  MoveL 1970 to (54.79, -51.67, -202.81) mm, rotated rx -11.83 ry -17.7 rz 126.62 deg; joints [4.443, -31.963, 116.112, 232.159, 70.658, -42.553, 143.741]
  MoveL 1971 to (53.18, -53.45, -205.23) mm, rotated rx -11.83 ry -17.7 rz 126.62 deg; joints [4.464, -31.726, 115.928, 232.166, 70.692, -42.511, 143.741]
  MoveL 1972 to (51.41, -54.45, -207.66) mm, rotated rx -11.83 ry -17.7 rz 126.62 deg; joints [4.497, -31.513, 115.805, 232.174, 70.75, -42.437, 143.741]
  MoveL 1973 to (50.67, -54.51, -208.61) mm, rotated rx -11.83 ry -17.7 rz 126.62 deg; joints [4.514, -31.44, 115.785, 232.177, 70.783, -42.394, 143.741]
  MoveL 1974 to (50.01, -54.27, -209.39) mm, rotated rx -11.83 ry -17.7 rz 126.62 deg; joints [4.532, -31.389, 115.791, 232.18, 70.82, -42.347, 143.741]
  MoveL 1975 to (49.72, -54.04, -209.71) mm, rotated rx -11.83 ry -17.7 rz 126.62 deg; joints [4.542, -31.372, 115.804, 232.181, 70.839, -42.322, 143.741]
  MoveL 1976 to (49.46, -53.74, -209.99) mm, rotated rx -11.83 ry -17.7 rz 126.62 deg; joints [4.551, -31.36, 115.824, 232.182, 70.859, -42.296, 143.741]
  MoveL 1977 to (48.99, -52.91, -210.43) mm, rotated rx -11.83 ry -17.7 rz 126.62 deg; joints [4.57, -31.353, 115.885, 232.183, 70.902, -42.242, 143.741]
  MoveL 1978 to (48.62, -51.78, -210.69) mm, rotated rx -11.83 ry -17.7 rz 126.62 deg; joints [4.59, -31.369, 115.972, 232.183, 70.948, -42.183, 143.741]
  MoveL 1979 to (48.34, -50.36, -210.77) mm, rotated rx -11.83 ry -17.7 rz 126.62 deg; joints [4.61, -31.406, 116.086, 232.182, 70.996, -42.12, 143.741]
  MoveL 1980 to (48.26, -49.84, -210.77) mm, rotated rx -11.83 ry -17.7 rz 126.62 deg; joints [4.616, -31.422, 116.128, 232.182, 71.013, -42.098, 143.741]
  MoveL 1981 to (48.22, -49.39, -210.74) mm, rotated rx -11.83 ry -17.7 rz 126.62 deg; joints [4.622, -31.438, 116.166, 232.182, 71.026, -42.081, 143.741]
  MoveL 1982 to (48.19, -48.96, -210.7) mm, rotated rx -11.83 ry -17.7 rz 126.62 deg; joints [4.627, -31.455, 116.201, 232.182, 71.038, -42.065, 143.741]
  MoveL 1983 to (48.17, -48.54, -210.64) mm, rotated rx -11.83 ry -17.7 rz 126.62 deg; joints [4.631, -31.472, 116.237, 232.181, 71.05, -42.05, 143.741]
  MoveL 1984 to (48.14, -48.09, -210.6) mm, rotated rx -11.83 ry -17.7 rz 126.62 deg; joints [4.636, -31.489, 116.274, 232.181, 71.062, -42.034, 143.741]
  MoveL 1985 to (48.07, -47.58, -210.58) mm, rotated rx -11.83 ry -17.7 rz 126.62 deg; joints [4.643, -31.506, 116.315, 232.181, 71.078, -42.013, 143.741]
  MoveL 1986 to (48, -47.06, -210.58) mm, rotated rx -11.83 ry -17.7 rz 126.62 deg; joints [4.649, -31.522, 116.357, 232.181, 71.095, -41.992, 143.741]
  MoveL 1987 to (47.93, -46.57, -210.58) mm, rotated rx -11.83 ry -17.7 rz 126.62 deg; joints [4.656, -31.538, 116.398, 232.18, 71.11, -41.972, 143.741]
  MoveL 1988 to (47.87, -46.1, -210.55) mm, rotated rx -11.83 ry -17.7 rz 126.62 deg; joints [4.662, -31.553, 116.436, 232.18, 71.124, -41.953, 143.741]
  MoveL 1989 to (47.84, -45.68, -210.5) mm, rotated rx -11.83 ry -17.7 rz 126.62 deg; joints [4.667, -31.57, 116.471, 232.181, 71.136, -41.938, 143.741]
  MoveL 1990 to (47.81, -45.25, -210.44) mm, rotated rx -11.83 ry -17.7 rz 126.62 deg; joints [4.672, -31.587, 116.506, 232.181, 71.147, -41.924, 143.741]
  MoveL 1991 to (47.77, -44.79, -210.38) mm, rotated rx -11.83 ry -17.7 rz 126.62 deg; joints [4.677, -31.606, 116.545, 232.181, 71.16, -41.907, 143.741]
  MoveL 1992 to (47.71, -44.18, -210.35) mm, rotated rx -11.83 ry -17.7 rz 126.62 deg; joints [4.685, -31.627, 116.595, 232.181, 71.178, -41.883, 143.741]
  MoveL 1993 to (47.63, -43.39, -210.33) mm, rotated rx -11.83 ry -17.7 rz 126.62 deg; joints [4.694, -31.653, 116.659, 232.18, 71.202, -41.852, 143.741]
  MoveL 1994 to (47.4, -41.84, -210.33) mm, rotated rx -11.83 ry -17.7 rz 126.62 deg; joints [4.715, -31.7, 116.785, 232.18, 71.252, -41.788, 143.741]
  MoveL 1995 to (47.29, -41.01, -210.3) mm, rotated rx -11.83 ry -17.7 rz 126.62 deg; joints [4.725, -31.728, 116.852, 232.18, 71.277, -41.755, 143.741]
  MoveL 1996 to (47.21, -40.39, -210.28) mm, rotated rx -11.83 ry -17.7 rz 126.62 deg; joints [4.733, -31.748, 116.903, 232.179, 71.296, -41.73, 143.741]
  MoveL 1997 to (47.19, -39.9, -210.28) mm, rotated rx -11.83 ry -17.7 rz 126.62 deg; joints [4.738, -31.764, 116.943, 232.178, 71.311, -41.71, 143.741]
  MoveL 1998 to (47.21, -39.48, -210.26) mm, rotated rx -11.83 ry -17.7 rz 126.62 deg; joints [4.74, -31.78, 116.978, 232.175, 71.323, -41.695, 143.741]
  MoveL 1999 to (47.26, -39.28, -210.15) mm, rotated rx -11.83 ry -17.7 rz 126.62 deg; joints [4.741, -31.794, 116.996, 232.175, 71.325, -41.691, 143.741]
  MoveL 2000 to (47.3, -39.34, -209.93) mm, rotated rx -11.83 ry -17.7 rz 126.62 deg; joints [4.742, -31.806, 116.993, 232.18, 71.316, -41.704, 143.741]
  MoveL 2001 to (47.32, -39.68, -209.58) mm, rotated rx -11.83 ry -17.7 rz 126.62 deg; joints [4.744, -31.814, 116.967, 232.191, 71.295, -41.733, 143.741]
  MoveL 2002 to (48.02, -39.34, -208.88) mm, rotated rx -11.83 ry -17.7 rz 126.62 deg; joints [4.726, -31.883, 117.01, 232.18, 71.278, -41.753, 143.741]
  MoveL 2003 to (48.92, -37.54, -208.73) mm, rotated rx -11.83 ry -17.7 rz 126.62 deg; joints [4.703, -31.975, 117.174, 232.138, 71.321, -41.692, 143.741]
  MoveL 2004 to (49.81, -35.84, -208.44) mm, rotated rx -11.83 ry -17.7 rz 126.62 deg; joints [4.682, -32.071, 117.33, 232.1, 71.357, -41.64, 143.741]
  MoveL 2005 to (50.69, -34.12, -208.17) mm, rotated rx -11.83 ry -17.7 rz 126.62 deg; joints [4.661, -32.166, 117.488, 232.062, 71.394, -41.587, 143.741]
  MoveL 2006 to (51.56, -32.39, -207.9) mm, rotated rx -11.83 ry -17.7 rz 126.62 deg; joints [4.641, -32.262, 117.646, 232.025, 71.431, -41.534, 143.741]
  MoveL 2007 to (52.46, -30.58, -207.68) mm, rotated rx -11.83 ry -17.7 rz 126.62 deg; joints [4.618, -32.358, 117.811, 231.984, 71.472, -41.476, 143.741]
  MoveL 2008 to (53.47, -28.71, -207.54) mm, rotated rx -11.83 ry -17.7 rz 126.62 deg; joints [4.591, -32.454, 117.981, 231.937, 71.516, -41.413, 143.741]
  MoveL 2009 to (54.76, -26.53, -207.43) mm, rotated rx -11.83 ry -17.7 rz 126.62 deg; joints [4.553, -32.566, 118.182, 231.875, 71.568, -41.337, 143.741]
  MoveL 2010 to (55.72, -24.23, -207.36) mm, rotated rx -11.83 ry -17.7 rz 126.62 deg; joints [4.53, -32.671, 118.386, 231.826, 71.628, -41.254, 143.741]
  MoveL 2011 to (56.53, -22.28, -207.24) mm, rotated rx -11.83 ry -17.7 rz 126.62 deg; joints [4.511, -32.764, 118.56, 231.785, 71.678, -41.186, 143.741]
  MoveL 2012 to (57.3, -20.55, -207.07) mm, rotated rx -11.83 ry -17.7 rz 126.62 deg; joints [4.493, -32.851, 118.715, 231.749, 71.718, -41.129, 143.741]
  MoveL 2013 to (58.17, -18.7, -206.94) mm, rotated rx -11.83 ry -17.7 rz 126.62 deg; joints [4.471, -32.942, 118.881, 231.708, 71.763, -41.066, 143.741]
  MoveL 2014 to (59.06, -16.82, -206.81) mm, rotated rx -11.83 ry -17.7 rz 126.62 deg; joints [4.448, -33.035, 119.05, 231.665, 71.809, -41.003, 143.741]
  MoveL 2015 to (59.99, -14.86, -206.74) mm, rotated rx -11.83 ry -17.7 rz 126.62 deg; joints [4.423, -33.128, 119.225, 231.618, 71.859, -40.933, 143.741]
  MoveL 2016 to (60.9, -12.92, -206.51) mm, rotated rx -11.83 ry -17.7 rz 126.62 deg; joints [4.401, -33.228, 119.398, 231.577, 71.903, -40.872, 143.741]
  MoveL 2017 to (61.8, -10.99, -206.4) mm, rotated rx -11.83 ry -17.7 rz 126.62 deg; joints [4.377, -33.322, 119.57, 231.533, 71.951, -40.806, 143.741]
  MoveL 2018 to (62.7, -9.06, -206.18) mm, rotated rx -11.83 ry -17.7 rz 126.62 deg; joints [4.356, -33.422, 119.743, 231.493, 71.995, -40.745, 143.741]
  MoveL 2019 to (63.6, -7.12, -206.07) mm, rotated rx -11.83 ry -17.7 rz 126.62 deg; joints [4.332, -33.515, 119.916, 231.449, 72.043, -40.68, 143.741]
  MoveL 2020 to (64.49, -5.18, -205.85) mm, rotated rx -11.83 ry -17.7 rz 126.62 deg; joints [4.311, -33.615, 120.088, 231.409, 72.088, -40.618, 143.741]
  MoveL 2021 to (65.39, -3.24, -205.74) mm, rotated rx -11.83 ry -17.7 rz 126.62 deg; joints [4.287, -33.708, 120.26, 231.365, 72.135, -40.553, 143.741]
  MoveL 2022 to (66.29, -1.3, -205.63) mm, rotated rx -11.83 ry -17.7 rz 126.62 deg; joints [4.263, -33.801, 120.432, 231.321, 72.184, -40.488, 143.741]
  MoveL 2023 to (67.04, 0.46, -205.4) mm, rotated rx -11.83 ry -17.7 rz 126.62 deg; joints [4.247, -33.891, 120.587, 231.288, 72.223, -40.434, 143.741]
  MoveL 2024 to (67.71, 2.16, -205.1) mm, rotated rx -11.83 ry -17.7 rz 126.62 deg; joints [4.233, -33.982, 120.737, 231.26, 72.259, -40.385, 143.741]
  MoveL 2025 to (68.34, 3.85, -204.71) mm, rotated rx -11.83 ry -17.7 rz 126.62 deg; joints [4.224, -34.077, 120.885, 231.237, 72.293, -40.341, 143.741]
  MoveL 2026 to (67.49, 2.71, -203.79) mm, rotated rx -11.83 ry -17.7 rz 126.62 deg; joints [4.266, -34.072, 120.784, 231.304, 72.234, -40.422, 143.741]
  MoveL 2027 to (67.66, 3.03, -203.73) mm, rotated rx -11.83 ry -17.7 rz 126.62 deg; joints [4.262, -34.091, 120.813, 231.297, 72.241, -40.413, 143.741]
  MoveL 2028 to (67.85, 3.35, -203.68) mm, rotated rx -11.83 ry -17.7 rz 126.62 deg; joints [4.256, -34.109, 120.842, 231.289, 72.247, -40.404, 143.741]
  MoveL 2029 to (68.13, 3.66, -203.64) mm, rotated rx -11.83 ry -17.7 rz 126.62 deg; joints [4.247, -34.129, 120.871, 231.277, 72.253, -40.396, 143.741]
  MoveL 2030 to (68.47, 3.95, -203.61) mm, rotated rx -11.83 ry -17.7 rz 126.62 deg; joints [4.234, -34.148, 120.9, 231.262, 72.258, -40.387, 143.741]
  MoveL 2031 to (68.89, 4.23, -203.61) mm, rotated rx -11.83 ry -17.7 rz 126.62 deg; joints [4.218, -34.168, 120.929, 231.244, 72.263, -40.38, 143.741]
  MoveL 2032 to (69.32, 4.5, -203.6) mm, rotated rx -11.83 ry -17.7 rz 126.62 deg; joints [4.202, -34.189, 120.958, 231.225, 72.267, -40.372, 143.741]
  MoveL 2033 to (70.23, 5.05, -203.6) mm, rotated rx -11.83 ry -17.7 rz 126.62 deg; joints [4.166, -34.229, 121.015, 231.185, 72.276, -40.357, 143.741]
  MoveL 2034 to (70.64, 5.31, -203.58) mm, rotated rx -11.83 ry -17.7 rz 126.62 deg; joints [4.15, -34.249, 121.042, 231.167, 72.28, -40.351, 143.741]
  MoveL 2035 to (71.03, 5.57, -203.54) mm, rotated rx -11.83 ry -17.7 rz 126.62 deg; joints [4.136, -34.27, 121.069, 231.151, 72.283, -40.346, 143.741]
  MoveL 2036 to (71.45, 5.88, -203.46) mm, rotated rx -11.83 ry -17.7 rz 126.62 deg; joints [4.121, -34.296, 121.101, 231.135, 72.286, -40.34, 143.741]
  MoveL 2037 to (71.92, 6.21, -203.39) mm, rotated rx -11.83 ry -17.7 rz 126.62 deg; joints [4.104, -34.323, 121.135, 231.115, 72.29, -40.333, 143.741]
  MoveL 2038 to (72.41, 6.53, -203.36) mm, rotated rx -11.83 ry -17.7 rz 126.62 deg; joints [4.086, -34.347, 121.167, 231.095, 72.294, -40.326, 143.741]
  MoveL 2039 to (72.87, 6.81, -203.35) mm, rotated rx -11.83 ry -17.7 rz 126.62 deg; joints [4.068, -34.368, 121.196, 231.075, 72.298, -40.319, 143.741]
  MoveL 2040 to (73.33, 7.08, -203.35) mm, rotated rx -11.83 ry -17.7 rz 126.62 deg; joints [4.05, -34.389, 121.225, 231.055, 72.303, -40.312, 143.741]
  MoveL 2041 to (74.23, 7.62, -203.35) mm, rotated rx -11.83 ry -17.7 rz 126.62 deg; joints [4.014, -34.429, 121.282, 231.015, 72.311, -40.297, 143.741]
  MoveL 2042 to (75.09, 8.17, -203.32) mm, rotated rx -11.83 ry -17.7 rz 126.62 deg; joints [3.981, -34.471, 121.339, 230.977, 72.32, -40.283, 143.741]
  MoveL 2043 to (77.35, 9.51, -203.32) mm, rotated rx -11.83 ry -17.7 rz 126.62 deg; joints [3.892, -34.571, 121.479, 230.878, 72.341, -40.248, 143.741]
  MoveL 2044 to (78.62, 10.19, -203.41) mm, rotated rx -11.83 ry -17.7 rz 126.62 deg; joints [3.84, -34.621, 121.551, 230.82, 72.353, -40.227, 143.741]
  MoveL 2045 to (79.73, 10.61, -203.67) mm, rotated rx -11.83 ry -17.7 rz 126.62 deg; joints [3.791, -34.646, 121.6, 230.765, 72.366, -40.207, 143.741]
  MoveL 2046 to (80.65, 10.77, -204.11) mm, rotated rx -11.83 ry -17.7 rz 126.62 deg; joints [3.746, -34.649, 121.623, 230.713, 72.377, -40.188, 143.741]
  MoveL 2047 to (81.05, 10.75, -204.39) mm, rotated rx -11.83 ry -17.7 rz 126.62 deg; joints [3.724, -34.641, 121.626, 230.689, 72.383, -40.179, 143.741]
  MoveL 2048 to (81.41, 10.67, -204.72) mm, rotated rx -11.83 ry -17.7 rz 126.62 deg; joints [3.703, -34.628, 121.623, 230.666, 72.389, -40.17, 143.741]
  MoveL 2049 to (81.98, 10.31, -205.51) mm, rotated rx -11.83 ry -17.7 rz 126.62 deg; joints [3.664, -34.583, 121.598, 230.621, 72.399, -40.153, 143.741]
  MoveL 2050 to (82.38, 9.68, -206.48) mm, rotated rx -11.83 ry -17.7 rz 126.62 deg; joints [3.629, -34.515, 121.549, 230.581, 72.41, -40.136, 143.741]
  MoveL 2051 to (82.66, 7.66, -208.93) mm, rotated rx -11.83 ry -17.7 rz 126.62 deg; joints [3.568, -34.309, 121.377, 230.511, 72.429, -40.107, 143.741]
  MoveL 2052 to (82.24, 5.27, -211.39) mm, rotated rx -11.83 ry -17.7 rz 126.62 deg; joints [3.535, -34.074, 121.165, 230.472, 72.443, -40.086, 143.741]
  MoveL 2053 to (81.1, 3.2, -213.14) mm, rotated rx -11.83 ry -17.7 rz 126.62 deg; joints [3.545, -33.874, 120.972, 230.481, 72.448, -40.081, 143.741]
  MoveL 2054 to (80.27, 2.28, -213.76) mm, rotated rx -11.83 ry -17.7 rz 126.62 deg; joints [3.567, -33.787, 120.883, 230.503, 72.448, -40.083, 143.741]
  MoveL 2055 to (79.26, 1.45, -214.2) mm, rotated rx -11.83 ry -17.7 rz 126.62 deg; joints [3.599, -33.708, 120.799, 230.537, 72.445, -40.089, 143.741]
  MoveL 2056 to (76.71, 0.01, -214.55) mm, rotated rx -11.83 ry -17.7 rz 126.62 deg; joints [3.695, -33.577, 120.645, 230.639, 72.434, -40.111, 143.741]
  MoveL 2057 to (74.29, -1.04, -214.54) mm, rotated rx -11.83 ry -17.7 rz 126.62 deg; joints [3.792, -33.483, 120.526, 230.744, 72.422, -40.135, 143.741]
  MoveL 2058 to (73.81, -1.24, -214.53) mm, rotated rx -11.83 ry -17.7 rz 126.62 deg; joints [3.812, -33.465, 120.502, 230.765, 72.419, -40.14, 143.741]
  MoveL 2059 to (73.31, -1.44, -214.5) mm, rotated rx -11.83 ry -17.7 rz 126.62 deg; joints [3.833, -33.448, 120.479, 230.787, 72.417, -40.145, 143.741]
  MoveL 2060 to (72.85, -1.63, -214.49) mm, rotated rx -11.83 ry -17.7 rz 126.62 deg; joints [3.851, -33.431, 120.457, 230.807, 72.414, -40.15, 143.741]
  MoveL 2061 to (72.44, -1.82, -214.51) mm, rotated rx -11.83 ry -17.7 rz 126.62 deg; joints [3.867, -33.413, 120.436, 230.824, 72.412, -40.154, 143.741]
  MoveL 2062 to (72, -2.03, -214.54) mm, rotated rx -11.83 ry -17.7 rz 126.62 deg; joints [3.884, -33.394, 120.412, 230.843, 72.41, -40.158, 143.741]
  MoveL 2063 to (71.49, -2.3, -214.61) mm, rotated rx -11.83 ry -17.7 rz 126.62 deg; joints [3.904, -33.368, 120.382, 230.863, 72.408, -40.162, 143.741]
  MoveL 2064 to (70.98, -2.58, -214.69) mm, rotated rx -11.83 ry -17.7 rz 126.62 deg; joints [3.922, -33.342, 120.352, 230.883, 72.407, -40.166, 143.741]
  MoveL 2065 to (70.48, -2.84, -214.73) mm, rotated rx -11.83 ry -17.7 rz 126.62 deg; joints [3.942, -33.318, 120.323, 230.904, 72.405, -40.17, 143.741]
  MoveL 2066 to (70, -3.07, -214.76) mm, rotated rx -11.83 ry -17.7 rz 126.62 deg; joints [3.961, -33.298, 120.298, 230.924, 72.402, -40.175, 143.741]
  MoveL 2067 to (69.52, -3.28, -214.77) mm, rotated rx -11.83 ry -17.7 rz 126.62 deg; joints [3.98, -33.278, 120.274, 230.944, 72.4, -40.18, 143.741]
  MoveL 2068 to (69.04, -3.49, -214.77) mm, rotated rx -11.83 ry -17.7 rz 126.62 deg; joints [3.999, -33.26, 120.25, 230.965, 72.397, -40.184, 143.741]
  MoveL 2069 to (68.54, -3.74, -214.8) mm, rotated rx -11.83 ry -17.7 rz 126.62 deg; joints [4.019, -33.237, 120.222, 230.986, 72.395, -40.189, 143.741]
  MoveL 2070 to (68.05, -4, -214.85) mm, rotated rx -11.83 ry -17.7 rz 126.62 deg; joints [4.037, -33.213, 120.193, 231.006, 72.393, -40.194, 143.741]
  MoveL 2071 to (67.57, -4.28, -214.92) mm, rotated rx -11.83 ry -17.7 rz 126.62 deg; joints [4.055, -33.188, 120.163, 231.025, 72.39, -40.199, 143.741]
  MoveL 2072 to (67.16, -4.58, -214.98) mm, rotated rx -11.83 ry -17.7 rz 126.62 deg; joints [4.07, -33.165, 120.132, 231.042, 72.386, -40.205, 143.741]
  MoveL 2073 to (66.81, -4.88, -215.01) mm, rotated rx -11.83 ry -17.7 rz 126.62 deg; joints [4.082, -33.144, 120.102, 231.057, 72.381, -40.214, 143.741]
  MoveL 2074 to (66.56, -5.19, -215.02) mm, rotated rx -11.83 ry -17.7 rz 126.62 deg; joints [4.091, -33.127, 120.073, 231.069, 72.373, -40.224, 143.741]
  MoveL 2075 to (66.33, -5.51, -215.02) mm, rotated rx -11.83 ry -17.7 rz 126.62 deg; joints [4.098, -33.111, 120.043, 231.08, 72.365, -40.235, 143.741]
  MoveL 2076 to (67.2, -4.56, -215.9) mm, rotated rx -11.83 ry -17.7 rz 126.62 deg; joints [4.055, -33.112, 120.129, 231.015, 72.417, -40.164, 143.741]
  MoveL 2077 to (66.44, -5.97, -216.18) mm, rotated rx -11.83 ry -17.7 rz 126.62 deg; joints [4.074, -33.031, 120.002, 231.046, 72.388, -40.203, 143.741]
  MoveL 2078 to (65.53, -7.53, -216.37) mm, rotated rx -11.83 ry -17.7 rz 126.62 deg; joints [4.099, -32.946, 119.86, 231.085, 72.354, -40.25, 143.741]
  MoveL 2079 to (64.47, -9.28, -216.51) mm, rotated rx -11.83 ry -17.7 rz 126.62 deg; joints [4.131, -32.854, 119.7, 231.135, 72.312, -40.307, 143.741]
  MoveL 2080 to (63.27, -11.18, -216.59) mm, rotated rx -11.83 ry -17.7 rz 126.62 deg; joints [4.169, -32.757, 119.526, 231.191, 72.266, -40.371, 143.741]
  MoveL 2081 to (62.15, -13, -216.74) mm, rotated rx -11.83 ry -17.7 rz 126.62 deg; joints [4.202, -32.661, 119.36, 231.242, 72.223, -40.429, 143.741]
  MoveL 2082 to (61.03, -14.82, -216.95) mm, rotated rx -11.83 ry -17.7 rz 126.62 deg; joints [4.234, -32.561, 119.193, 231.292, 72.183, -40.486, 143.741]
  MoveL 2083 to (59.96, -16.55, -217.08) mm, rotated rx -11.83 ry -17.7 rz 126.62 deg; joints [4.266, -32.47, 119.034, 231.341, 72.142, -40.543, 143.741]
  MoveL 2084 to (59.01, -18.13, -217.34) mm, rotated rx -11.83 ry -17.7 rz 126.62 deg; joints [4.292, -32.379, 118.888, 231.382, 72.109, -40.589, 143.741]
  MoveL 2085 to (57.92, -19.89, -217.56) mm, rotated rx -11.83 ry -17.7 rz 126.62 deg; joints [4.324, -32.282, 118.727, 231.429, 72.07, -40.643, 143.741]
  MoveL 2086 to (56.81, -21.65, -217.7) mm, rotated rx -11.83 ry -17.7 rz 126.62 deg; joints [4.357, -32.188, 118.564, 231.48, 72.029, -40.701, 143.741]
  MoveL 2087 to (55.66, -23.45, -217.8) mm, rotated rx -11.83 ry -17.7 rz 126.62 deg; joints [4.391, -32.094, 118.397, 231.534, 71.985, -40.762, 143.741]
  MoveL 2088 to (54.53, -25.25, -218.03) mm, rotated rx -11.83 ry -17.7 rz 126.62 deg; joints [4.423, -31.994, 118.231, 231.583, 71.946, -40.818, 143.741]
  MoveL 2089 to (53.37, -27.05, -218.29) mm, rotated rx -11.83 ry -17.7 rz 126.62 deg; joints [4.457, -31.89, 118.063, 231.633, 71.907, -40.873, 143.741]
  MoveL 2090 to (52.22, -28.84, -218.38) mm, rotated rx -11.83 ry -17.7 rz 126.62 deg; joints [4.491, -31.798, 117.897, 231.687, 71.864, -40.935, 143.741]
  MoveL 2091 to (51.05, -30.67, -218.42) mm, rotated rx -11.83 ry -17.7 rz 126.62 deg; joints [4.528, -31.705, 117.727, 231.744, 71.818, -41, 143.741]
  MoveL 2092 to (49.9, -32.45, -218.53) mm, rotated rx -11.83 ry -17.7 rz 126.62 deg; joints [4.562, -31.612, 117.562, 231.797, 71.775, -41.061, 143.741]
  MoveL 2093 to (48.75, -34.22, -218.73) mm, rotated rx -11.83 ry -17.7 rz 126.62 deg; joints [4.595, -31.513, 117.395, 231.848, 71.735, -41.119, 143.741]
  MoveL 2094 to (47.6, -35.96, -219.06) mm, rotated rx -11.83 ry -17.7 rz 126.62 deg; joints [4.627, -31.408, 117.232, 231.895, 71.701, -41.169, 143.741]
  MoveL 2095 to (46.4, -37.75, -219.32) mm, rotated rx -11.83 ry -17.7 rz 126.62 deg; joints [4.661, -31.304, 117.063, 231.947, 71.663, -41.224, 143.741]
  MoveL 2096 to (45.21, -39.52, -219.52) mm, rotated rx -11.83 ry -17.7 rz 126.62 deg; joints [4.695, -31.204, 116.896, 231.999, 71.624, -41.281, 143.741]
  MoveL 2097 to (43.98, -41.32, -219.76) mm, rotated rx -11.83 ry -17.7 rz 126.62 deg; joints [4.731, -31.1, 116.725, 232.052, 71.585, -41.339, 143.741]
  MoveL 2098 to (42.8, -43.11, -219.9) mm, rotated rx -11.83 ry -17.7 rz 126.62 deg; joints [4.766, -31.003, 116.556, 232.107, 71.543, -41.4, 143.741]
  MoveL 2099 to (41.65, -44.89, -219.93) mm, rotated rx -11.83 ry -17.7 rz 126.62 deg; joints [4.8, -30.914, 116.389, 232.163, 71.497, -41.467, 143.741]
  MoveL 2100 to (41.06, -45.13, -220.59) mm, rotated rx -11.83 ry -17.7 rz 126.62 deg; joints [4.814, -30.854, 116.356, 232.169, 71.515, -41.445, 143.741]
  MoveL 2101 to (41.16, -44.81, -220.92) mm, rotated rx -11.83 ry -17.7 rz 126.62 deg; joints [4.808, -30.848, 116.382, 232.154, 71.534, -41.418, 143.741]
  MoveL 2102 to (41.17, -44.77, -221.13) mm, rotated rx -11.83 ry -17.7 rz 126.62 deg; joints [4.805, -30.838, 116.385, 232.148, 71.541, -41.407, 143.741]
  MoveL 2103 to (41.1, -44.97, -221.23) mm, rotated rx -11.83 ry -17.7 rz 126.62 deg; joints [4.805, -30.824, 116.366, 232.15, 71.539, -41.411, 143.741]
  MoveL 2104 to (41.02, -45.39, -221.25) mm, rotated rx -11.83 ry -17.7 rz 126.62 deg; joints [4.805, -30.807, 116.33, 232.155, 71.527, -41.427, 143.741]
  MoveC 2105 to (40.97, -46.4, -221.25) mm, rotated rx -11.83 ry -17.7 rz 126.62 deg; joints [4.8, -30.771, 116.245, 232.162, 71.496, -41.468, 143.741] to (41, -47.42, -221.25) mm, rotated rx -11.83 ry -17.7 rz 126.62 deg; joints [4.792, -30.738, 116.16, 232.168, 71.464, -41.51, 143.741]
  MoveL 2106 to (41, -47.42, -221.25) mm, rotated rx -11.83 ry -17.7 rz 126.62 deg; joints [4.792, -30.737, 116.16, 232.167, 71.464, -41.51, 143.741]
  MoveL 2107 to (41, -47.96, -221.28) mm, rotated rx -11.83 ry -17.7 rz 126.62 deg; joints [4.787, -30.718, 116.115, 232.17, 71.448, -41.531, 143.741]
  MoveL 2108 to (40.98, -48.5, -221.33) mm, rotated rx -11.83 ry -17.7 rz 126.62 deg; joints [4.784, -30.696, 116.069, 232.173, 71.433, -41.551, 143.741]
  MoveL 2109 to (40.95, -49.08, -221.4) mm, rotated rx -11.83 ry -17.7 rz 126.62 deg; joints [4.78, -30.672, 116.02, 232.176, 71.417, -41.572, 143.741]
  MoveL 2110 to (40.93, -49.68, -221.44) mm, rotated rx -11.83 ry -17.7 rz 126.62 deg; joints [4.776, -30.65, 115.97, 232.179, 71.4, -41.595, 143.741]
  MoveL 2111 to (40.94, -50.89, -221.46) mm, rotated rx -11.83 ry -17.7 rz 126.62 deg; joints [4.767, -30.608, 115.868, 232.185, 71.363, -41.644, 143.741]
  MoveL 2112 to (40.93, -51.45, -221.49) mm, rotated rx -11.83 ry -17.7 rz 126.62 deg; joints [4.763, -30.587, 115.821, 232.188, 71.347, -41.665, 143.741]
  MoveL 2113 to (40.89, -51.92, -221.56) mm, rotated rx -11.83 ry -17.7 rz 126.62 deg; joints [4.76, -30.566, 115.781, 232.191, 71.335, -41.682, 143.741]
  MoveL 2114 to (40.85, -52.35, -221.65) mm, rotated rx -11.83 ry -17.7 rz 126.62 deg; joints [4.757, -30.545, 115.743, 232.193, 71.324, -41.695, 143.741]
  MoveL 2115 to (40.82, -52.78, -221.72) mm, rotated rx -11.83 ry -17.7 rz 126.62 deg; joints [4.755, -30.526, 115.707, 232.195, 71.313, -41.71, 143.741]
  MoveL 2116 to (40.81, -53.23, -221.75) mm, rotated rx -11.83 ry -17.7 rz 126.62 deg; joints [4.752, -30.509, 115.669, 232.197, 71.3, -41.727, 143.741]
  MoveL 2117 to (40.86, -55.85, -221.75) mm, rotated rx -11.83 ry -17.7 rz 126.62 deg; joints [4.731, -30.421, 115.45, 232.211, 71.219, -41.835, 143.741]
  MoveL 2118 to (40.66, -58.75, -222.1) mm, rotated rx -11.83 ry -17.7 rz 126.62 deg; joints [4.714, -30.298, 115.201, 232.228, 71.14, -41.939, 143.741]
  MoveL 2119 to (40.35, -59.99, -222.53) mm, rotated rx -11.83 ry -17.7 rz 126.62 deg; joints [4.713, -30.224, 115.089, 232.237, 71.117, -41.971, 143.741]
  MoveL 2120 to (39.89, -61.1, -223.13) mm, rotated rx -11.83 ry -17.7 rz 126.62 deg; joints [4.715, -30.142, 114.985, 232.245, 71.104, -41.989, 143.741]
  MoveL 2121 to (39.3, -62.07, -223.91) mm, rotated rx -11.83 ry -17.7 rz 126.62 deg; joints [4.722, -30.051, 114.889, 232.254, 71.101, -41.994, 143.741]
  MoveL 2122 to (38.57, -62.9, -224.86) mm, rotated rx -11.83 ry -17.7 rz 126.62 deg; joints [4.734, -29.952, 114.802, 232.262, 71.109, -41.985, 143.741]
  MoveL 2123 to (36.7, -64.16, -227.27) mm, rotated rx -11.83 ry -17.7 rz 126.62 deg; joints [4.77, -29.729, 114.65, 232.279, 71.155, -41.927, 143.741]
  MoveL 2124 to (34.85, -64.63, -229.68) mm, rotated rx -11.83 ry -17.7 rz 126.62 deg; joints [4.809, -29.534, 114.566, 232.29, 71.226, -41.837, 143.741]
  MoveL 2125 to (34.16, -64.47, -230.63) mm, rotated rx -11.83 ry -17.7 rz 126.62 deg; joints [4.826, -29.47, 114.561, 232.291, 71.264, -41.788, 143.741]
  MoveL 2126 to (33.62, -64.06, -231.41) mm, rotated rx -11.83 ry -17.7 rz 126.62 deg; joints [4.841, -29.427, 114.582, 232.289, 71.303, -41.736, 143.741]
  MoveL 2127 to (33.41, -63.75, -231.73) mm, rotated rx -11.83 ry -17.7 rz 126.62 deg; joints [4.847, -29.414, 114.602, 232.286, 71.324, -41.709, 143.741]
  MoveL 2128 to (33.24, -63.38, -232.01) mm, rotated rx -11.83 ry -17.7 rz 126.62 deg; joints [4.853, -29.407, 114.629, 232.283, 71.345, -41.681, 143.741]
  MoveL 2129 to (33.01, -62.45, -232.44) mm, rotated rx -11.83 ry -17.7 rz 126.62 deg; joints [4.863, -29.408, 114.7, 232.275, 71.389, -41.623, 143.741]
  MoveL 2130 to (32.94, -61.26, -232.7) mm, rotated rx -11.83 ry -17.7 rz 126.62 deg; joints [4.871, -29.432, 114.798, 232.263, 71.434, -41.562, 143.741]
  MoveL 2131 to (33.02, -59.81, -232.79) mm, rotated rx -11.83 ry -17.7 rz 126.62 deg; joints [4.877, -29.478, 114.92, 232.249, 71.482, -41.498, 143.741]
  MoveL 2132 to (33.07, -59.29, -232.79) mm, rotated rx -11.83 ry -17.7 rz 126.62 deg; joints [4.879, -29.496, 114.965, 232.243, 71.498, -41.476, 143.741]
  MoveL 2133 to (33.13, -58.84, -232.75) mm, rotated rx -11.83 ry -17.7 rz 126.62 deg; joints [4.88, -29.515, 115.004, 232.239, 71.51, -41.459, 143.741]
  MoveL 2134 to (33.21, -58.43, -232.7) mm, rotated rx -11.83 ry -17.7 rz 126.62 deg; joints [4.88, -29.533, 115.04, 232.235, 71.521, -41.445, 143.741]
  MoveL 2135 to (33.29, -58.03, -232.63) mm, rotated rx -11.83 ry -17.7 rz 126.62 deg; joints [4.88, -29.553, 115.075, 232.231, 71.531, -41.431, 143.741]
  MoveL 2136 to (33.37, -57.59, -232.58) mm, rotated rx -11.83 ry -17.7 rz 126.62 deg; joints [4.881, -29.572, 115.114, 232.227, 71.543, -41.415, 143.741]
  MoveL 2137 to (33.43, -57.09, -232.56) mm, rotated rx -11.83 ry -17.7 rz 126.62 deg; joints [4.882, -29.591, 115.157, 232.222, 71.558, -41.395, 143.741]
  MoveL 2138 to (34, -51.39, -232.55) mm, rotated rx -11.83 ry -17.7 rz 126.62 deg; joints [4.9, -29.795, 115.644, 232.165, 71.732, -41.161, 143.741]
  MoveL 2139 to (34.09, -50.63, -232.54) mm, rotated rx -11.83 ry -17.7 rz 126.62 deg; joints [4.901, -29.823, 115.709, 232.157, 71.755, -41.13, 143.741]
  MoveL 2140 to (34.19, -49.98, -232.53) mm, rotated rx -11.83 ry -17.7 rz 126.62 deg; joints [4.902, -29.847, 115.765, 232.149, 71.774, -41.104, 143.741]
  MoveL 2141 to (34.37, -49.43, -232.52) mm, rotated rx -11.83 ry -17.7 rz 126.62 deg; joints [4.898, -29.87, 115.814, 232.139, 71.79, -41.082, 143.741]
  MoveL 2142 to (34.61, -48.95, -232.48) mm, rotated rx -11.83 ry -17.7 rz 126.62 deg; joints [4.893, -29.895, 115.858, 232.128, 71.802, -41.065, 143.741]
  MoveL 2143 to (34.8, -48.68, -232.32) mm, rotated rx -11.83 ry -17.7 rz 126.62 deg; joints [4.889, -29.917, 115.885, 232.123, 71.804, -41.061, 143.741]
  MoveL 2144 to (34.82, -48.69, -232.01) mm, rotated rx -11.83 ry -17.7 rz 126.62 deg; joints [4.892, -29.935, 115.886, 232.131, 71.795, -41.075, 143.741]
  MoveL 2145 to (34.65, -49.02, -231.53) mm, rotated rx -11.83 ry -17.7 rz 126.62 deg; joints [4.904, -29.948, 115.86, 232.152, 71.771, -41.108, 143.741]
  MoveL 2146 to (35.27, -49.11, -230.55) mm, rotated rx -11.83 ry -17.7 rz 126.62 deg; joints [4.89, -30.015, 115.869, 232.154, 71.735, -41.156, 143.741]
  MoveL 2147 to (36.49, -47.69, -230.25) mm, rotated rx -11.83 ry -17.7 rz 126.62 deg; joints [4.854, -30.109, 116.009, 232.105, 71.761, -41.116, 143.741]
  MoveL 2148 to (37.77, -46.2, -230.05) mm, rotated rx -11.83 ry -17.7 rz 126.62 deg; joints [4.814, -30.201, 116.156, 232.051, 71.792, -41.069, 143.741]
  MoveL 2149 to (39.13, -44.57, -229.92) mm, rotated rx -11.83 ry -17.7 rz 126.62 deg; joints [4.77, -30.295, 116.315, 231.99, 71.83, -41.013, 143.741]
  MoveL 2150 to (41.85, -41.28, -229.92) mm, rotated rx -11.83 ry -17.7 rz 126.62 deg; joints [4.68, -30.47, 116.633, 231.862, 71.913, -40.891, 143.741]
  MoveL 2151 to (43.11, -39.75, -229.83) mm, rotated rx -11.83 ry -17.7 rz 126.62 deg; joints [4.639, -30.556, 116.781, 231.804, 71.949, -40.838, 143.741]
  MoveL 2152 to (44.47, -38.1, -229.83) mm, rotated rx -11.83 ry -17.7 rz 126.62 deg; joints [4.594, -30.644, 116.939, 231.74, 71.991, -40.777, 143.741]
  MoveL 2153 to (45.92, -36.5, -229.83) mm, rotated rx -11.83 ry -17.7 rz 126.62 deg; joints [4.544, -30.732, 117.095, 231.673, 72.03, -40.719, 143.741]
  MoveL 2154 to (47.65, -34.64, -229.65) mm, rotated rx -11.83 ry -17.7 rz 126.62 deg; joints [4.486, -30.846, 117.278, 231.597, 72.07, -40.66, 143.741]
  MoveL 2155 to (48.97, -32.84, -229.42) mm, rotated rx -11.83 ry -17.7 rz 126.62 deg; joints [4.447, -30.95, 117.449, 231.54, 72.11, -40.603, 143.741]
  MoveL 2156 to (50.27, -31.11, -229.3) mm, rotated rx -11.83 ry -17.7 rz 126.62 deg; joints [4.405, -31.046, 117.614, 231.481, 72.151, -40.545, 143.741]
  MoveL 2157 to (51.63, -29.46, -229.19) mm, rotated rx -11.83 ry -17.7 rz 126.62 deg; joints [4.361, -31.139, 117.772, 231.419, 72.189, -40.49, 143.741]
  MoveL 2158 to (52.98, -27.81, -228.98) mm, rotated rx -11.83 ry -17.7 rz 126.62 deg; joints [4.318, -31.239, 117.931, 231.361, 72.224, -40.44, 143.741]
  MoveL 2159 to (54.33, -26.16, -228.87) mm, rotated rx -11.83 ry -17.7 rz 126.62 deg; joints [4.273, -31.332, 118.089, 231.3, 72.263, -40.385, 143.741]
  MoveL 2160 to (55.68, -24.51, -228.76) mm, rotated rx -11.83 ry -17.7 rz 126.62 deg; joints [4.229, -31.425, 118.246, 231.239, 72.301, -40.331, 143.741]
  MoveL 2161 to (57.02, -22.85, -228.55) mm, rotated rx -11.83 ry -17.7 rz 126.62 deg; joints [4.186, -31.524, 118.405, 231.181, 72.336, -40.28, 143.741]
  MoveL 2162 to (58.37, -21.19, -228.44) mm, rotated rx -11.83 ry -17.7 rz 126.62 deg; joints [4.141, -31.617, 118.562, 231.12, 72.375, -40.226, 143.741]
  MoveL 2163 to (59.71, -19.54, -228.34) mm, rotated rx -11.83 ry -17.7 rz 126.62 deg; joints [4.097, -31.71, 118.719, 231.059, 72.413, -40.172, 143.741]
  MoveL 2164 to (61.04, -17.87, -228.13) mm, rotated rx -11.83 ry -17.7 rz 126.62 deg; joints [4.054, -31.809, 118.878, 231.002, 72.449, -40.122, 143.741]
  MoveL 2165 to (62.39, -16.21, -228.03) mm, rotated rx -11.83 ry -17.7 rz 126.62 deg; joints [4.009, -31.902, 119.035, 230.941, 72.488, -40.068, 143.741]
  MoveL 2166 to (63.49, -14.72, -227.77) mm, rotated rx -11.83 ry -17.7 rz 126.62 deg; joints [3.976, -31.992, 119.174, 230.895, 72.518, -40.027, 143.741]
  MoveL 2167 to (64.44, -13.35, -227.41) mm, rotated rx -11.83 ry -17.7 rz 126.62 deg; joints [3.949, -32.081, 119.303, 230.858, 72.542, -39.994, 143.741]
  MoveL 2168 to (65.25, -12.06, -226.9) mm, rotated rx -11.83 ry -17.7 rz 126.62 deg; joints [3.931, -32.173, 119.425, 230.832, 72.56, -39.969, 143.741]
  MoveL 2169 to (64.35, -12.75, -226.06) mm, rotated rx -11.83 ry -17.7 rz 126.62 deg; joints [3.977, -32.178, 119.36, 230.896, 72.517, -40.027, 143.741]
  MoveL 2170 to (64.56, -12.5, -226.03) mm, rotated rx -11.83 ry -17.7 rz 126.62 deg; joints [3.97, -32.193, 119.383, 230.886, 72.523, -40.02, 143.741]
  MoveL 2171 to (64.79, -12.27, -225.99) mm, rotated rx -11.83 ry -17.7 rz 126.62 deg; joints [3.962, -32.208, 119.406, 230.877, 72.527, -40.014, 143.741]
  MoveL 2172 to (65.1, -12.08, -225.93) mm, rotated rx -11.83 ry -17.7 rz 126.62 deg; joints [3.95, -32.225, 119.427, 230.865, 72.529, -40.011, 143.741]
  MoveL 2173 to (65.48, -11.9, -225.9) mm, rotated rx -11.83 ry -17.7 rz 126.62 deg; joints [3.936, -32.243, 119.447, 230.849, 72.53, -40.008, 143.741]
  MoveL 2174 to (65.94, -11.73, -225.87) mm, rotated rx -11.83 ry -17.7 rz 126.62 deg; joints [3.918, -32.261, 119.467, 230.831, 72.531, -40.005, 143.741]
  MoveL 2175 to (70.45, -10.38, -225.87) mm, rotated rx -11.83 ry -17.7 rz 126.62 deg; joints [3.733, -32.416, 119.644, 230.639, 72.537, -39.982, 143.741]
  MoveL 2176 to (70.83, -10.25, -225.85) mm, rotated rx -11.83 ry -17.7 rz 126.62 deg; joints [3.718, -32.431, 119.661, 230.623, 72.538, -39.98, 143.741]
  MoveL 2177 to (71.33, -10.1, -225.85) mm, rotated rx -11.83 ry -17.7 rz 126.62 deg; joints [3.697, -32.448, 119.68, 230.602, 72.539, -39.978, 143.741]
  MoveL 2178 to (72.31, -9.78, -225.81) mm, rotated rx -11.83 ry -17.7 rz 126.62 deg; joints [3.658, -32.485, 119.721, 230.561, 72.539, -39.974, 143.741]
  MoveL 2179 to (74.82, -9.03, -225.81) mm, rotated rx -11.83 ry -17.7 rz 126.62 deg; joints [3.555, -32.571, 119.818, 230.455, 72.543, -39.961, 143.741]
  MoveL 2180 to (75.79, -8.67, -225.79) mm, rotated rx -11.83 ry -17.7 rz 126.62 deg; joints [3.516, -32.607, 119.86, 230.414, 72.545, -39.955, 143.741]
  MoveL 2181 to (77.17, -8.24, -225.86) mm, rotated rx -11.83 ry -17.7 rz 126.62 deg; joints [3.458, -32.651, 119.915, 230.353, 72.55, -39.945, 143.741]
  MoveL 2182 to (78.32, -8.03, -226.11) mm, rotated rx -11.83 ry -17.7 rz 126.62 deg; joints [3.406, -32.672, 119.946, 230.298, 72.555, -39.934, 143.741]
  MoveL 2183 to (79.25, -8.04, -226.55) mm, rotated rx -11.83 ry -17.7 rz 126.62 deg; joints [3.36, -32.668, 119.956, 230.248, 72.562, -39.922, 143.741]
  MoveL 2184 to (79.63, -8.13, -226.84) mm, rotated rx -11.83 ry -17.7 rz 126.62 deg; joints [3.339, -32.657, 119.952, 230.225, 72.565, -39.916, 143.741]
  MoveL 2185 to (79.95, -8.27, -227.17) mm, rotated rx -11.83 ry -17.7 rz 126.62 deg; joints [3.319, -32.641, 119.943, 230.203, 72.569, -39.909, 143.741]
  MoveL 2186 to (80.43, -8.72, -227.99) mm, rotated rx -11.83 ry -17.7 rz 126.62 deg; joints [3.284, -32.59, 119.908, 230.164, 72.578, -39.896, 143.741]
  MoveL 2187 to (80.68, -9.39, -228.98) mm, rotated rx -11.83 ry -17.7 rz 126.62 deg; joints [3.254, -32.516, 119.85, 230.13, 72.588, -39.881, 143.741]
  MoveL 2188 to (80.51, -11.4, -231.54) mm, rotated rx -11.83 ry -17.7 rz 126.62 deg; joints [3.212, -32.296, 119.667, 230.079, 72.61, -39.85, 143.741]
  MoveL 2189 to (79.58, -13.61, -234.11) mm, rotated rx -11.83 ry -17.7 rz 126.62 deg; joints [3.202, -32.05, 119.456, 230.06, 72.631, -39.822, 143.741]
  MoveL 2190 to (78.02, -15.35, -235.94) mm, rotated rx -11.83 ry -17.7 rz 126.62 deg; joints [3.232, -31.848, 119.279, 230.084, 72.649, -39.803, 143.741]
  MoveL 2191 to (77, -16.04, -236.58) mm, rotated rx -11.83 ry -17.7 rz 126.62 deg; joints [3.262, -31.764, 119.204, 230.112, 72.656, -39.796, 143.741]
  MoveL 2192 to (75.83, -16.61, -237.04) mm, rotated rx -11.83 ry -17.7 rz 126.62 deg; joints [3.302, -31.69, 119.138, 230.151, 72.662, -39.791, 143.741]
  MoveL 2193 to (73.02, -17.39, -237.4) mm, rotated rx -11.83 ry -17.7 rz 126.62 deg; joints [3.412, -31.574, 119.031, 230.26, 72.671, -39.788, 143.741]
  MoveL 2194 to (69.92, -17.93, -237.4) mm, rotated rx -11.83 ry -17.7 rz 126.62 deg; joints [3.542, -31.481, 118.942, 230.39, 72.678, -39.788, 143.741]
  MoveL 2195 to (68.92, -18.13, -237.42) mm, rotated rx -11.83 ry -17.7 rz 126.62 deg; joints [3.583, -31.45, 118.911, 230.431, 72.68, -39.789, 143.741]
  MoveL 2196 to (67.89, -18.31, -237.42) mm, rotated rx -11.83 ry -17.7 rz 126.62 deg; joints [3.626, -31.419, 118.881, 230.474, 72.682, -39.789, 143.741]
  MoveL 2197 to (67.4, -18.4, -237.42) mm, rotated rx -11.83 ry -17.7 rz 126.62 deg; joints [3.646, -31.403, 118.866, 230.494, 72.683, -39.789, 143.741]
  MoveL 2198 to (66.75, -18.52, -237.45) mm, rotated rx -11.83 ry -17.7 rz 126.62 deg; joints [3.673, -31.382, 118.846, 230.521, 72.685, -39.789, 143.741]
  MoveL 2199 to (66.17, -18.66, -237.51) mm, rotated rx -11.83 ry -17.7 rz 126.62 deg; joints [3.696, -31.36, 118.826, 230.544, 72.687, -39.788, 143.741]
  MoveL 2200 to (65.68, -18.79, -237.58) mm, rotated rx -11.83 ry -17.7 rz 126.62 deg; joints [3.715, -31.34, 118.808, 230.562, 72.689, -39.787, 143.741]
  MoveL 2201 to (65.23, -18.9, -237.63) mm, rotated rx -11.83 ry -17.7 rz 126.62 deg; joints [3.733, -31.322, 118.792, 230.58, 72.691, -39.786, 143.741]
  MoveL 2202 to (64.78, -19, -237.67) mm, rotated rx -11.83 ry -17.7 rz 126.62 deg; joints [3.751, -31.306, 118.777, 230.598, 72.692, -39.786, 143.741]
  MoveL 2203 to (63.23, -19.27, -237.67) mm, rotated rx -11.83 ry -17.7 rz 126.62 deg; joints [3.816, -31.259, 118.731, 230.663, 72.695, -39.787, 143.741]
  MoveL 2204 to (62.74, -19.38, -237.68) mm, rotated rx -11.83 ry -17.7 rz 126.62 deg; joints [3.836, -31.243, 118.715, 230.683, 72.696, -39.787, 143.741]
  MoveL 2205 to (62.31, -19.49, -237.71) mm, rotated rx -11.83 ry -17.7 rz 126.62 deg; joints [3.853, -31.227, 118.699, 230.7, 72.696, -39.788, 143.741]
  MoveL 2206 to (61.95, -19.62, -237.75) mm, rotated rx -11.83 ry -17.7 rz 126.62 deg; joints [3.867, -31.211, 118.683, 230.715, 72.696, -39.789, 143.741]
  MoveL 2207 to (61.69, -19.78, -237.82) mm, rotated rx -11.83 ry -17.7 rz 126.62 deg; joints [3.876, -31.196, 118.665, 230.724, 72.695, -39.791, 143.741]
  MoveL 2208 to (61.48, -19.96, -237.89) mm, rotated rx -11.83 ry -17.7 rz 126.62 deg; joints [3.882, -31.181, 118.647, 230.732, 72.693, -39.794, 143.741]
  MoveL 2209 to (62.99, -19.46, -238.69) mm, rotated rx -11.83 ry -17.7 rz 126.62 deg; joints [3.81, -31.187, 118.705, 230.646, 72.724, -39.749, 143.741]
  MoveL 2210 to (61.69, -20.65, -239.1) mm, rotated rx -11.83 ry -17.7 rz 126.62 deg; joints [3.852, -31.093, 118.584, 230.695, 72.708, -39.773, 143.741]
  MoveL 2211 to (60.33, -21.94, -239.36) mm, rotated rx -11.83 ry -17.7 rz 126.62 deg; joints [3.898, -31.003, 118.456, 230.75, 72.686, -39.805, 143.741]
  MoveL 2212 to (58.89, -23.33, -239.54) mm, rotated rx -11.83 ry -17.7 rz 126.62 deg; joints [3.947, -30.913, 118.318, 230.812, 72.657, -39.845, 143.741]
  MoveL 2213 to (57.37, -24.83, -239.74) mm, rotated rx -11.83 ry -17.7 rz 126.62 deg; joints [3.999, -30.817, 118.17, 230.877, 72.627, -39.888, 143.741]
  MoveL 2214 to (55.84, -26.32, -239.83) mm, rotated rx -11.83 ry -17.7 rz 126.62 deg; joints [4.053, -30.726, 118.024, 230.945, 72.593, -39.936, 143.741]
  MoveL 2215 to (54.31, -27.8, -239.93) mm, rotated rx -11.83 ry -17.7 rz 126.62 deg; joints [4.107, -30.635, 117.877, 231.013, 72.56, -39.983, 143.741]
  MoveL 2216 to (52.78, -29.3, -240.13) mm, rotated rx -11.83 ry -17.7 rz 126.62 deg; joints [4.159, -30.538, 117.729, 231.078, 72.529, -40.027, 143.741]
  MoveL 2217 to (51.24, -30.78, -240.23) mm, rotated rx -11.83 ry -17.7 rz 126.62 deg; joints [4.213, -30.448, 117.581, 231.146, 72.496, -40.074, 143.741]
  MoveL 2218 to (49.71, -32.26, -240.33) mm, rotated rx -11.83 ry -17.7 rz 126.62 deg; joints [4.266, -30.357, 117.434, 231.214, 72.463, -40.122, 143.741]
  MoveL 2219 to (48.17, -33.74, -240.53) mm, rotated rx -11.83 ry -17.7 rz 126.62 deg; joints [4.318, -30.26, 117.286, 231.279, 72.433, -40.166, 143.741]
  MoveL 2220 to (45.09, -36.7, -240.73) mm, rotated rx -11.83 ry -17.7 rz 126.62 deg; joints [4.425, -30.078, 116.991, 231.415, 72.366, -40.263, 143.741]
  MoveL 2221 to (43.8, -37.93, -240.94) mm, rotated rx -11.83 ry -17.7 rz 126.62 deg; joints [4.468, -29.994, 116.866, 231.469, 72.342, -40.298, 143.741]
  MoveL 2222 to (42.41, -39.32, -241.01) mm, rotated rx -11.83 ry -17.7 rz 126.62 deg; joints [4.516, -29.912, 116.728, 231.531, 72.31, -40.345, 143.741]
  MoveL 2223 to (40.99, -40.81, -241.02) mm, rotated rx -11.83 ry -17.7 rz 126.62 deg; joints [4.565, -29.828, 116.581, 231.596, 72.273, -40.399, 143.741]
  MoveL 2224 to (39.05, -42.65, -241.13) mm, rotated rx -11.83 ry -17.7 rz 126.62 deg; joints [4.632, -29.715, 116.396, 231.682, 72.231, -40.461, 143.741]
  MoveL 2225 to (37.1, -44.34, -241.22) mm, rotated rx -11.83 ry -17.7 rz 126.62 deg; joints [4.701, -29.608, 116.222, 231.767, 72.194, -40.518, 143.741]
  MoveL 2226 to (35.47, -45.83, -241.32) mm, rotated rx -11.83 ry -17.7 rz 126.62 deg; joints [4.757, -29.514, 116.07, 231.839, 72.16, -40.568, 143.741]
  MoveL 2227 to (33.98, -47.23, -241.49) mm, rotated rx -11.83 ry -17.7 rz 126.62 deg; joints [4.807, -29.422, 115.928, 231.903, 72.131, -40.612, 143.741]
  MoveL 2228 to (32.58, -48.52, -241.77) mm, rotated rx -11.83 ry -17.7 rz 126.62 deg; joints [4.853, -29.33, 115.794, 231.959, 72.108, -40.648, 143.741]
  MoveL 2229 to (31.18, -49.8, -242.06) mm, rotated rx -11.83 ry -17.7 rz 126.62 deg; joints [4.898, -29.238, 115.662, 232.015, 72.085, -40.683, 143.741]
  MoveL 2230 to (29.77, -51.05, -242.35) mm, rotated rx -11.83 ry -17.7 rz 126.62 deg; joints [4.944, -29.147, 115.532, 232.071, 72.064, -40.717, 143.741]
  MoveL 2231 to (28.31, -52.39, -242.51) mm, rotated rx -11.83 ry -17.7 rz 126.62 deg; joints [4.993, -29.058, 115.393, 232.133, 72.035, -40.761, 143.741]
  MoveL 2232 to (27.66, -52.39, -243.13) mm, rotated rx -11.83 ry -17.7 rz 126.62 deg; joints [5.011, -29.007, 115.378, 232.143, 72.058, -40.732, 143.741]
  MoveL 2233 to (27.77, -52.09, -243.44) mm, rotated rx -11.83 ry -17.7 rz 126.62 deg; joints [5.005, -29.002, 115.403, 232.129, 72.076, -40.707, 143.741]
  MoveL 2234 to (27.74, -52.05, -243.63) mm, rotated rx -11.83 ry -17.7 rz 126.62 deg; joints [5.004, -28.992, 115.404, 232.125, 72.083, -40.697, 143.741]
  MoveL 2235 to (27.6, -52.26, -243.73) mm, rotated rx -11.83 ry -17.7 rz 126.62 deg; joints [5.007, -28.976, 115.383, 232.129, 72.08, -40.701, 143.741]
  MoveL 2236 to (27.42, -52.67, -243.75) mm, rotated rx -11.83 ry -17.7 rz 126.62 deg; joints [5.011, -28.957, 115.346, 232.138, 72.069, -40.717, 143.741]
  MoveL 2237 to (27.26, -53.13, -243.75) mm, rotated rx -11.83 ry -17.7 rz 126.62 deg; joints [5.014, -28.938, 115.305, 232.147, 72.056, -40.736, 143.741]
  MoveL 2238 to (27.05, -54.08, -243.78) mm, rotated rx -11.83 ry -17.7 rz 126.62 deg; joints [5.016, -28.9, 115.221, 232.16, 72.028, -40.774, 143.741]
  MoveL 2239 to (26.71, -55.62, -243.78) mm, rotated rx -11.83 ry -17.7 rz 126.62 deg; joints [5.019, -28.842, 115.087, 232.183, 71.981, -40.837, 143.741]
  MoveL 2240 to (26.46, -56.56, -243.8) mm, rotated rx -11.83 ry -17.7 rz 126.62 deg; joints [5.022, -28.804, 115.003, 232.198, 71.953, -40.875, 143.741]
  MoveL 2241 to (26.24, -57.59, -243.8) mm, rotated rx -11.83 ry -17.7 rz 126.62 deg; joints [5.024, -28.765, 114.913, 232.213, 71.922, -40.917, 143.741]
  MoveL 2242 to (26.12, -58.09, -243.82) mm, rotated rx -11.83 ry -17.7 rz 126.62 deg; joints [5.025, -28.745, 114.869, 232.22, 71.908, -40.938, 143.741]
  MoveL 2243 to (26, -58.55, -243.85) mm, rotated rx -11.83 ry -17.7 rz 126.62 deg; joints [5.026, -28.726, 114.829, 232.226, 71.895, -40.955, 143.741]
  MoveL 2244 to (25.89, -58.97, -243.89) mm, rotated rx -11.83 ry -17.7 rz 126.62 deg; joints [5.027, -28.706, 114.791, 232.232, 71.883, -40.971, 143.741]
  MoveL 2245 to (25.77, -59.36, -243.95) mm, rotated rx -11.83 ry -17.7 rz 126.62 deg; joints [5.028, -28.687, 114.756, 232.238, 71.874, -40.984, 143.741]
  MoveL 2246 to (25.66, -59.76, -244.01) mm, rotated rx -11.83 ry -17.7 rz 126.62 deg; joints [5.029, -28.668, 114.72, 232.243, 71.863, -40.998, 143.741]
  MoveL 2247 to (25.54, -60.21, -244.04) mm, rotated rx -11.83 ry -17.7 rz 126.62 deg; joints [5.03, -28.649, 114.68, 232.25, 71.851, -41.015, 143.741]
  MoveL 2248 to (25.42, -60.67, -244.07) mm, rotated rx -11.83 ry -17.7 rz 126.62 deg; joints [5.031, -28.63, 114.639, 232.257, 71.838, -41.033, 143.741]
  MoveL 2249 to (25.3, -61.09, -244.11) mm, rotated rx -11.83 ry -17.7 rz 126.62 deg; joints [5.033, -28.61, 114.601, 232.263, 71.826, -41.049, 143.741]
  MoveL 2250 to (25.18, -61.47, -244.17) mm, rotated rx -11.83 ry -17.7 rz 126.62 deg; joints [5.034, -28.591, 114.566, 232.269, 71.817, -41.062, 143.741]
  MoveL 2251 to (25.06, -61.86, -244.22) mm, rotated rx -11.83 ry -17.7 rz 126.62 deg; joints [5.036, -28.573, 114.531, 232.274, 71.807, -41.076, 143.741]
  MoveL 2252 to (24.94, -62.29, -244.25) mm, rotated rx -11.83 ry -17.7 rz 126.62 deg; joints [5.037, -28.554, 114.493, 232.281, 71.795, -41.092, 143.741]
  MoveL 2253 to (24.83, -62.8, -244.25) mm, rotated rx -11.83 ry -17.7 rz 126.62 deg; joints [5.038, -28.535, 114.448, 232.288, 71.779, -41.114, 143.741]
  MoveL 2254 to (23.95, -65.58, -244.61) mm, rotated rx -11.83 ry -17.7 rz 126.62 deg; joints [5.049, -28.402, 114.196, 232.331, 71.707, -41.213, 143.741]
  MoveL 2255 to (23.38, -66.74, -245.05) mm, rotated rx -11.83 ry -17.7 rz 126.62 deg; joints [5.059, -28.325, 114.085, 232.349, 71.687, -41.242, 143.741]
  MoveL 2256 to (22.7, -67.73, -245.68) mm, rotated rx -11.83 ry -17.7 rz 126.62 deg; joints [5.071, -28.241, 113.985, 232.366, 71.678, -41.256, 143.741]
  MoveL 2257 to (21.07, -69.24, -247.46) mm, rotated rx -11.83 ry -17.7 rz 126.62 deg; joints [5.103, -28.052, 113.816, 232.393, 71.692, -41.241, 143.741]
  MoveL 2258 to (19.06, -70.11, -249.95) mm, rotated rx -11.83 ry -17.7 rz 126.62 deg; joints [5.146, -27.835, 113.687, 232.413, 71.748, -41.169, 143.741]
  MoveL 2259 to (17.27, -70.21, -252.44) mm, rotated rx -11.83 ry -17.7 rz 126.62 deg; joints [5.185, -27.648, 113.626, 232.42, 71.827, -41.066, 143.741]
  MoveL 2260 to (16.67, -69.93, -253.42) mm, rotated rx -11.83 ry -17.7 rz 126.62 deg; joints [5.198, -27.587, 113.631, 232.417, 71.868, -41.012, 143.741]
  MoveL 2261 to (16.28, -69.43, -254.22) mm, rotated rx -11.83 ry -17.7 rz 126.62 deg; joints [5.207, -27.549, 113.659, 232.408, 71.909, -40.957, 143.741]
  MoveL 2262 to (16.16, -69.1, -254.56) mm, rotated rx -11.83 ry -17.7 rz 126.62 deg; joints [5.21, -27.538, 113.683, 232.403, 71.93, -40.929, 143.741]
  MoveL 2263 to (16.09, -68.71, -254.85) mm, rotated rx -11.83 ry -17.7 rz 126.62 deg; joints [5.212, -27.533, 113.712, 232.396, 71.951, -40.9, 143.741]
  MoveL 2264 to (16.1, -67.76, -255.29) mm, rotated rx -11.83 ry -17.7 rz 126.62 deg; joints [5.213, -27.539, 113.788, 232.378, 71.994, -40.842, 143.741]
  MoveL 2265 to (16.31, -66.59, -255.56) mm, rotated rx -11.83 ry -17.7 rz 126.62 deg; joints [5.209, -27.567, 113.888, 232.356, 72.038, -40.781, 143.741]
  MoveL 2266 to (16.73, -65.2, -255.65) mm, rotated rx -11.83 ry -17.7 rz 126.62 deg; joints [5.201, -27.617, 114.012, 232.328, 72.082, -40.72, 143.741]
  MoveL 2267 to (17.58, -62.72, -255.65) mm, rotated rx -11.83 ry -17.7 rz 126.62 deg; joints [5.184, -27.717, 114.235, 232.28, 72.157, -40.617, 143.741]
  MoveL 2268 to (17.73, -62.31, -255.62) mm, rotated rx -11.83 ry -17.7 rz 126.62 deg; joints [5.181, -27.736, 114.273, 232.272, 72.168, -40.601, 143.741]
  MoveL 2269 to (17.89, -61.94, -255.57) mm, rotated rx -11.83 ry -17.7 rz 126.62 deg; joints [5.178, -27.755, 114.307, 232.265, 72.178, -40.588, 143.741]
  MoveL 2270 to (18.04, -61.59, -255.5) mm, rotated rx -11.83 ry -17.7 rz 126.62 deg; joints [5.175, -27.774, 114.34, 232.258, 72.186, -40.576, 143.741]
  MoveL 2271 to (18.21, -61.19, -255.45) mm, rotated rx -11.83 ry -17.7 rz 126.62 deg; joints [5.172, -27.793, 114.377, 232.251, 72.196, -40.562, 143.741]
  MoveL 2272 to (18.39, -60.72, -255.41) mm, rotated rx -11.83 ry -17.7 rz 126.62 deg; joints [5.168, -27.815, 114.419, 232.242, 72.209, -40.544, 143.741]
  MoveL 2273 to (18.59, -60.24, -255.35) mm, rotated rx -11.83 ry -17.7 rz 126.62 deg; joints [5.164, -27.838, 114.464, 232.233, 72.222, -40.526, 143.741]
  MoveL 2274 to (18.77, -59.73, -255.34) mm, rotated rx -11.83 ry -17.7 rz 126.62 deg; joints [5.16, -27.86, 114.51, 232.223, 72.237, -40.506, 143.741]
  MoveL 2275 to (18.98, -59.12, -255.35) mm, rotated rx -11.83 ry -17.7 rz 126.62 deg; joints [5.156, -27.884, 114.565, 232.211, 72.255, -40.48, 143.741]
  MoveL 2276 to (19.23, -58.29, -255.42) mm, rotated rx -11.83 ry -17.7 rz 126.62 deg; joints [5.151, -27.913, 114.638, 232.194, 72.282, -40.443, 143.741]
  MoveL 2277 to (19.4, -57.79, -255.42) mm, rotated rx -11.83 ry -17.7 rz 126.62 deg; joints [5.147, -27.933, 114.683, 232.184, 72.297, -40.423, 143.741]
  MoveL 2278 to (19.57, -57.32, -255.41) mm, rotated rx -11.83 ry -17.7 rz 126.62 deg; joints [5.144, -27.952, 114.725, 232.175, 72.311, -40.403, 143.741]
  MoveL 2279 to (19.73, -56.88, -255.39) mm, rotated rx -11.83 ry -17.7 rz 126.62 deg; joints [5.141, -27.972, 114.765, 232.167, 72.324, -40.386, 143.741]
  MoveL 2280 to (19.89, -56.5, -255.34) mm, rotated rx -11.83 ry -17.7 rz 126.62 deg; joints [5.138, -27.991, 114.801, 232.159, 72.334, -40.373, 143.741]
  MoveL 2281 to (20.06, -56.14, -255.28) mm, rotated rx -11.83 ry -17.7 rz 126.62 deg; joints [5.134, -28.01, 114.834, 232.152, 72.342, -40.36, 143.741]
  MoveL 2282 to (20.28, -55.78, -255.23) mm, rotated rx -11.83 ry -17.7 rz 126.62 deg; joints [5.128, -28.029, 114.869, 232.143, 72.351, -40.348, 143.741]
  MoveL 2283 to (20.53, -55.45, -255.17) mm, rotated rx -11.83 ry -17.7 rz 126.62 deg; joints [5.121, -28.049, 114.901, 232.132, 72.359, -40.337, 143.741]
  MoveL 2284 to (20.71, -55.32, -255.01) mm, rotated rx -11.83 ry -17.7 rz 126.62 deg; joints [5.117, -28.067, 114.917, 232.128, 72.357, -40.339, 143.741]
  MoveL 2285 to (20.71, -55.43, -254.7) mm, rotated rx -11.83 ry -17.7 rz 126.62 deg; joints [5.12, -28.081, 114.91, 232.137, 72.344, -40.356, 143.741]
  MoveL 2286 to (20.51, -55.82, -254.21) mm, rotated rx -11.83 ry -17.7 rz 126.62 deg; joints [5.133, -28.092, 114.878, 232.16, 72.319, -40.392, 143.741]
  MoveL 2287 to (21.19, -55.25, -253.35) mm, rotated rx -11.83 ry -17.7 rz 126.62 deg; joints [5.12, -28.175, 114.945, 232.152, 72.308, -40.406, 143.741]
  MoveL 2288 to (24.59, -52.67, -253.35) mm, rotated rx -11.83 ry -17.7 rz 126.62 deg; joints [4.997, -28.341, 115.22, 232, 72.37, -40.31, 143.741]
  MoveL 2289 to (26.18, -51.46, -253.29) mm, rotated rx -11.83 ry -17.7 rz 126.62 deg; joints [4.94, -28.422, 115.349, 231.931, 72.397, -40.269, 143.741]
  MoveL 2290 to (27.78, -50.27, -253.14) mm, rotated rx -11.83 ry -17.7 rz 126.62 deg; joints [4.884, -28.507, 115.477, 231.863, 72.421, -40.232, 143.741]
  MoveL 2291 to (29.62, -48.9, -252.94) mm, rotated rx -11.83 ry -17.7 rz 126.62 deg; joints [4.82, -28.607, 115.624, 231.787, 72.448, -40.19, 143.741]
  MoveL 2292 to (31.36, -47.6, -252.73) mm, rotated rx -11.83 ry -17.7 rz 126.62 deg; joints [4.759, -28.703, 115.764, 231.715, 72.472, -40.152, 143.741]
  MoveL 2293 to (33.1, -46.28, -252.63) mm, rotated rx -11.83 ry -17.7 rz 126.62 deg; joints [4.697, -28.793, 115.904, 231.64, 72.501, -40.109, 143.741]
  MoveL 2294 to (34.8, -44.99, -252.63) mm, rotated rx -11.83 ry -17.7 rz 126.62 deg; joints [4.635, -28.876, 116.04, 231.564, 72.531, -40.063, 143.741]
  MoveL 2295 to (36.38, -43.79, -252.56) mm, rotated rx -11.83 ry -17.7 rz 126.62 deg; joints [4.578, -28.956, 116.167, 231.495, 72.558, -40.023, 143.741]
  MoveL 2296 to (37.87, -42.65, -252.45) mm, rotated rx -11.83 ry -17.7 rz 126.62 deg; joints [4.525, -29.035, 116.287, 231.431, 72.582, -39.988, 143.741]
  MoveL 2297 to (39.49, -41.41, -252.38) mm, rotated rx -11.83 ry -17.7 rz 126.62 deg; joints [4.466, -29.118, 116.417, 231.36, 72.609, -39.947, 143.741]
  MoveL 2298 to (41.19, -40.12, -252.2) mm, rotated rx -11.83 ry -17.7 rz 126.62 deg; joints [4.406, -29.211, 116.554, 231.289, 72.634, -39.91, 143.741]
  MoveL 2299 to (44.58, -37.53, -252.02) mm, rotated rx -11.83 ry -17.7 rz 126.62 deg; joints [4.283, -29.386, 116.825, 231.142, 72.69, -39.827, 143.741]
  MoveL 2300 to (46.28, -36.23, -251.84) mm, rotated rx -11.83 ry -17.7 rz 126.62 deg; joints [4.223, -29.479, 116.962, 231.071, 72.716, -39.79, 143.741]
  MoveL 2301 to (47.97, -34.92, -251.66) mm, rotated rx -11.83 ry -17.7 rz 126.62 deg; joints [4.163, -29.572, 117.098, 230.999, 72.741, -39.753, 143.741]
  MoveL 2302 to (49.66, -33.63, -251.66) mm, rotated rx -11.83 ry -17.7 rz 126.62 deg; joints [4.099, -29.654, 117.232, 230.923, 72.771, -39.709, 143.741]
  MoveL 2303 to (51.35, -32.32, -251.48) mm, rotated rx -11.83 ry -17.7 rz 126.62 deg; joints [4.039, -29.747, 117.368, 230.852, 72.797, -39.672, 143.741]
  MoveL 2304 to (53.03, -31.01, -251.3) mm, rotated rx -11.83 ry -17.7 rz 126.62 deg; joints [3.979, -29.839, 117.505, 230.781, 72.823, -39.635, 143.741]
  MoveL 2305 to (54.73, -29.72, -251.3) mm, rotated rx -11.83 ry -17.7 rz 126.62 deg; joints [3.915, -29.921, 117.638, 230.704, 72.853, -39.592, 143.741]
  MoveL 2306 to (56.24, -28.48, -251.11) mm, rotated rx -11.83 ry -17.7 rz 126.62 deg; joints [3.862, -30.009, 117.765, 230.642, 72.877, -39.558, 143.741]
  MoveL 2307 to (57.52, -27.34, -250.79) mm, rotated rx -11.83 ry -17.7 rz 126.62 deg; joints [3.819, -30.094, 117.881, 230.591, 72.894, -39.533, 143.741]
  MoveL 2308 to (58.6, -26.27, -250.32) mm, rotated rx -11.83 ry -17.7 rz 126.62 deg; joints [3.787, -30.182, 117.99, 230.553, 72.907, -39.515, 143.741]
  MoveL 2309 to (57.76, -26.69, -249.56) mm, rotated rx -11.83 ry -17.7 rz 126.62 deg; joints [3.831, -30.193, 117.948, 230.61, 72.875, -39.558, 143.741]
  MoveL 2310 to (58.11, -26.48, -249.55) mm, rotated rx -11.83 ry -17.7 rz 126.62 deg; joints [3.817, -30.208, 117.971, 230.595, 72.879, -39.552, 143.741]
  MoveC 2311 to (61.63, -25.98, -249.55) mm, rotated rx -11.83 ry -17.7 rz 126.62 deg; joints [3.67, -30.31, 118.065, 230.449, 72.87, -39.554, 143.741] to (65.18, -25.78, -249.55) mm, rotated rx -11.83 ry -17.7 rz 126.62 deg; joints [3.52, -30.403, 118.135, 230.303, 72.851, -39.569, 143.741]
  MoveL 2312 to (65.18, -25.78, -249.55) mm, rotated rx -11.83 ry -17.7 rz 126.62 deg; joints [3.52, -30.403, 118.135, 230.303, 72.851, -39.569, 143.741]
  MoveL 2313 to (65.65, -25.74, -249.53) mm, rotated rx -11.83 ry -17.7 rz 126.62 deg; joints [3.501, -30.417, 118.146, 230.284, 72.848, -39.571, 143.741]
  MoveL 2314 to (66.07, -25.69, -249.48) mm, rotated rx -11.83 ry -17.7 rz 126.62 deg; joints [3.484, -30.432, 118.157, 230.268, 72.845, -39.574, 143.741]
  MoveL 2315 to (66.47, -25.63, -249.42) mm, rotated rx -11.83 ry -17.7 rz 126.62 deg; joints [3.468, -30.447, 118.168, 230.253, 72.842, -39.576, 143.741]
  MoveL 2316 to (66.91, -25.58, -249.37) mm, rotated rx -11.83 ry -17.7 rz 126.62 deg; joints [3.45, -30.462, 118.179, 230.236, 72.839, -39.579, 143.741]
  MoveL 2317 to (67.38, -25.53, -249.34) mm, rotated rx -11.83 ry -17.7 rz 126.62 deg; joints [3.431, -30.476, 118.19, 230.218, 72.836, -39.582, 143.741]
  MoveL 2318 to (67.89, -25.49, -249.33) mm, rotated rx -11.83 ry -17.7 rz 126.62 deg; joints [3.409, -30.491, 118.2, 230.197, 72.833, -39.584, 143.741]
  MoveL 2319 to (68.94, -25.43, -249.33) mm, rotated rx -11.83 ry -17.7 rz 126.62 deg; joints [3.365, -30.518, 118.221, 230.154, 72.827, -39.588, 143.741]
  MoveL 2320 to (70.4, -25.4, -249.42) mm, rotated rx -11.83 ry -17.7 rz 126.62 deg; joints [3.302, -30.549, 118.244, 230.092, 72.82, -39.593, 143.741]
  MoveL 2321 to (71.59, -25.5, -249.69) mm, rotated rx -11.83 ry -17.7 rz 126.62 deg; joints [3.246, -30.559, 118.251, 230.037, 72.816, -39.594, 143.741]
  MoveL 2322 to (72.53, -25.73, -250.15) mm, rotated rx -11.83 ry -17.7 rz 126.62 deg; joints [3.198, -30.548, 118.241, 229.988, 72.816, -39.591, 143.741]
  MoveL 2323 to (73.21, -26.09, -250.79) mm, rotated rx -11.83 ry -17.7 rz 126.62 deg; joints [3.158, -30.515, 118.216, 229.945, 72.82, -39.584, 143.741]
  MoveL 2324 to (73.64, -26.58, -251.61) mm, rotated rx -11.83 ry -17.7 rz 126.62 deg; joints [3.125, -30.462, 118.175, 229.909, 72.827, -39.573, 143.741]
  MoveL 2325 to (73.8, -27.21, -252.62) mm, rotated rx -11.83 ry -17.7 rz 126.62 deg; joints [3.099, -30.387, 118.118, 229.88, 72.837, -39.558, 143.741]
  MoveL 2326 to (73.35, -28.84, -255.18) mm, rotated rx -11.83 ry -17.7 rz 126.62 deg; joints [3.072, -30.175, 117.956, 229.84, 72.869, -39.518, 143.741]
  MoveL 2327 to (72.12, -30.47, -257.74) mm, rotated rx -11.83 ry -17.7 rz 126.62 deg; joints [3.078, -29.943, 117.781, 229.833, 72.906, -39.472, 143.741]
  MoveL 2328 to (71.29, -31.1, -258.74) mm, rotated rx -11.83 ry -17.7 rz 126.62 deg; joints [3.095, -29.845, 117.709, 229.844, 72.923, -39.452, 143.741]
  MoveL 2329 to (70.33, -31.6, -259.57) mm, rotated rx -11.83 ry -17.7 rz 126.62 deg; joints [3.121, -29.758, 117.646, 229.864, 72.94, -39.433, 143.741]
  MoveL 2330 to (69.22, -31.97, -260.21) mm, rotated rx -11.83 ry -17.7 rz 126.62 deg; joints [3.157, -29.682, 117.594, 229.895, 72.956, -39.415, 143.741]
  MoveL 2331 to (67.98, -32.21, -260.66) mm, rotated rx -11.83 ry -17.7 rz 126.62 deg; joints [3.202, -29.617, 117.552, 229.935, 72.971, -39.398, 143.741]
  MoveL 2332 to (65.09, -32.31, -261.03) mm, rotated rx -11.83 ry -17.7 rz 126.62 deg; joints [3.319, -29.523, 117.497, 230.043, 73, -39.369, 143.741]
  MoveL 2333 to (64.04, -32.26, -261.03) mm, rotated rx -11.83 ry -17.7 rz 126.62 deg; joints [3.364, -29.499, 117.486, 230.086, 73.01, -39.36, 143.741]
  MoveL 2334 to (63.52, -32.24, -261.04) mm, rotated rx -11.83 ry -17.7 rz 126.62 deg; joints [3.386, -29.487, 117.48, 230.107, 73.014, -39.355, 143.741]
  MoveL 2335 to (63.04, -32.23, -261.06) mm, rotated rx -11.83 ry -17.7 rz 126.62 deg; joints [3.406, -29.474, 117.473, 230.125, 73.019, -39.351, 143.741]
  MoveL 2336 to (62.62, -32.23, -261.11) mm, rotated rx -11.83 ry -17.7 rz 126.62 deg; joints [3.423, -29.461, 117.466, 230.141, 73.023, -39.347, 143.741]
  MoveL 2337 to (62.22, -32.24, -261.16) mm, rotated rx -11.83 ry -17.7 rz 126.62 deg; joints [3.44, -29.447, 117.459, 230.156, 73.027, -39.342, 143.741]
  MoveL 2338 to (61.8, -32.25, -261.21) mm, rotated rx -11.83 ry -17.7 rz 126.62 deg; joints [3.457, -29.434, 117.451, 230.172, 73.031, -39.338, 143.741]
  MoveL 2339 to (61.33, -32.24, -261.23) mm, rotated rx -11.83 ry -17.7 rz 126.62 deg; joints [3.477, -29.422, 117.445, 230.191, 73.036, -39.334, 143.741]
  MoveL 2340 to (60.83, -32.22, -261.24) mm, rotated rx -11.83 ry -17.7 rz 126.62 deg; joints [3.498, -29.41, 117.439, 230.211, 73.04, -39.329, 143.741]
  MoveL 2341 to (60.28, -32.19, -261.23) mm, rotated rx -11.83 ry -17.7 rz 126.62 deg; joints [3.522, -29.398, 117.433, 230.233, 73.045, -39.325, 143.741]
  MoveL 2342 to (59.75, -32.17, -261.24) mm, rotated rx -11.83 ry -17.7 rz 126.62 deg; joints [3.544, -29.385, 117.427, 230.254, 73.049, -39.32, 143.741]
  MoveL 2343 to (59.25, -32.15, -261.27) mm, rotated rx -11.83 ry -17.7 rz 126.62 deg; joints [3.565, -29.372, 117.42, 230.274, 73.054, -39.316, 143.741]
  MoveL 2344 to (58.78, -32.15, -261.31) mm, rotated rx -11.83 ry -17.7 rz 126.62 deg; joints [3.584, -29.358, 117.413, 230.292, 73.059, -39.311, 143.741]
  MoveL 2345 to (58.28, -32.16, -261.39) mm, rotated rx -11.83 ry -17.7 rz 126.62 deg; joints [3.605, -29.341, 117.403, 230.31, 73.064, -39.305, 143.741]
  MoveL 2346 to (57.67, -32.17, -261.45) mm, rotated rx -11.83 ry -17.7 rz 126.62 deg; joints [3.63, -29.322, 117.393, 230.333, 73.07, -39.299, 143.741]
  MoveL 2347 to (57.1, -32.16, -261.47) mm, rotated rx -11.83 ry -17.7 rz 126.62 deg; joints [3.654, -29.308, 117.385, 230.356, 73.075, -39.294, 143.741]
  MoveL 2348 to (56.57, -32.13, -261.47) mm, rotated rx -11.83 ry -17.7 rz 126.62 deg; joints [3.676, -29.296, 117.379, 230.377, 73.079, -39.29, 143.741]
  MoveL 2349 to (56.05, -32.11, -261.47) mm, rotated rx -11.83 ry -17.7 rz 126.62 deg; joints [3.699, -29.284, 117.373, 230.399, 73.084, -39.286, 143.741]
  MoveL 2350 to (55.39, -32.1, -261.48) mm, rotated rx -11.83 ry -17.7 rz 126.62 deg; joints [3.727, -29.268, 117.364, 230.425, 73.089, -39.281, 143.741]
  MoveL 2351 to (54.81, -32.11, -261.49) mm, rotated rx -11.83 ry -17.7 rz 126.62 deg; joints [3.751, -29.253, 117.354, 230.449, 73.093, -39.277, 143.741]
  MoveL 2352 to (54.3, -32.14, -261.5) mm, rotated rx -11.83 ry -17.7 rz 126.62 deg; joints [3.772, -29.239, 117.343, 230.469, 73.095, -39.275, 143.741]
  MoveL 2353 to (53.97, -32.22, -261.5) mm, rotated rx -11.83 ry -17.7 rz 126.62 deg; joints [3.786, -29.228, 117.331, 230.483, 73.095, -39.276, 143.741]
  MoveL 2354 to (53.72, -32.32, -261.5) mm, rotated rx -11.83 ry -17.7 rz 126.62 deg; joints [3.796, -29.219, 117.319, 230.494, 73.093, -39.279, 143.741]
  MoveL 2355 to (54.58, -31.95, -262.09) mm, rotated rx -11.83 ry -17.7 rz 126.62 deg; joints [3.753, -29.217, 117.358, 230.441, 73.118, -39.245, 143.741]
  MoveL 2356 to (53.6, -32.86, -262.62) mm, rotated rx -11.83 ry -17.7 rz 126.62 deg; joints [3.782, -29.134, 117.262, 230.473, 73.111, -39.255, 143.741]
  MoveL 2357 to (52.36, -33.81, -263) mm, rotated rx -11.83 ry -17.7 rz 126.62 deg; joints [3.823, -29.052, 117.161, 230.519, 73.1, -39.272, 143.741]
  MoveL 2358 to (50.84, -34.85, -263.26) mm, rotated rx -11.83 ry -17.7 rz 126.62 deg; joints [3.877, -28.967, 117.048, 230.58, 73.083, -39.296, 143.741]
  MoveL 2359 to (49.09, -35.94, -263.39) mm, rotated rx -11.83 ry -17.7 rz 126.62 deg; joints [3.942, -28.884, 116.93, 230.654, 73.063, -39.326, 143.741]
  MoveL 2360 to (47.3, -37.03, -263.48) mm, rotated rx -11.83 ry -17.7 rz 126.62 deg; joints [4.01, -28.801, 116.809, 230.73, 73.041, -39.358, 143.741]
  MoveL 2361 to (43.65, -39.25, -263.66) mm, rotated rx -11.83 ry -17.7 rz 126.62 deg; joints [4.147, -28.633, 116.565, 230.886, 72.996, -39.423, 143.741]
  MoveL 2362 to (41.83, -40.36, -263.84) mm, rotated rx -11.83 ry -17.7 rz 126.62 deg; joints [4.214, -28.544, 116.442, 230.962, 72.977, -39.452, 143.741]
  MoveL 2363 to (38.18, -42.57, -264.02) mm, rotated rx -11.83 ry -17.7 rz 126.62 deg; joints [4.35, -28.376, 116.197, 231.118, 72.932, -39.518, 143.741]
  MoveL 2364 to (36.36, -43.68, -264.2) mm, rotated rx -11.83 ry -17.7 rz 126.62 deg; joints [4.417, -28.286, 116.073, 231.193, 72.912, -39.548, 143.741]
  MoveL 2365 to (34.53, -44.78, -264.29) mm, rotated rx -11.83 ry -17.7 rz 126.62 deg; joints [4.485, -28.202, 115.95, 231.271, 72.89, -39.581, 143.741]
  MoveL 2366 to (32.83, -45.78, -264.5) mm, rotated rx -11.83 ry -17.7 rz 126.62 deg; joints [4.547, -28.118, 115.836, 231.34, 72.874, -39.607, 143.741]
  MoveL 2367 to (30.81, -46.99, -264.65) mm, rotated rx -11.83 ry -17.7 rz 126.62 deg; joints [4.621, -28.022, 115.699, 231.425, 72.851, -39.642, 143.741]
  MoveL 2368 to (28.61, -48.32, -264.77) mm, rotated rx -11.83 ry -17.7 rz 126.62 deg; joints [4.703, -27.921, 115.55, 231.518, 72.824, -39.683, 143.741]
  MoveL 2369 to (26.78, -49.42, -264.77) mm, rotated rx -11.83 ry -17.7 rz 126.62 deg; joints [4.771, -27.842, 115.427, 231.599, 72.798, -39.721, 143.741]
  MoveL 2370 to (25.04, -50.46, -264.84) mm, rotated rx -11.83 ry -17.7 rz 126.62 deg; joints [4.836, -27.762, 115.31, 231.673, 72.777, -39.755, 143.741]
  MoveL 2371 to (23.46, -51.38, -265.02) mm, rotated rx -11.83 ry -17.7 rz 126.62 deg; joints [4.893, -27.685, 115.203, 231.738, 72.761, -39.78, 143.741]
  MoveL 2372 to (21.84, -52.32, -265.23) mm, rotated rx -11.83 ry -17.7 rz 126.62 deg; joints [4.952, -27.604, 115.095, 231.803, 72.746, -39.804, 143.741]
  MoveL 2373 to (19.81, -53.52, -265.37) mm, rotated rx -11.83 ry -17.7 rz 126.62 deg; joints [5.026, -27.509, 114.958, 231.888, 72.722, -39.842, 143.741]
  MoveL 2374 to (17.59, -54.84, -265.47) mm, rotated rx -11.83 ry -17.7 rz 126.62 deg; joints [5.107, -27.408, 114.807, 231.982, 72.694, -39.885, 143.741]
  MoveL 2375 to (13.94, -57.04, -265.47) mm, rotated rx -11.83 ry -17.7 rz 126.62 deg; joints [5.243, -27.25, 114.557, 232.142, 72.643, -39.964, 143.741]
  MoveL 2376 to (13.63, -56.95, -266.17) mm, rotated rx -11.83 ry -17.7 rz 126.62 deg; joints [5.247, -27.206, 114.553, 232.136, 72.668, -39.931, 143.741]
  MoveL 2377 to (13.82, -56.7, -266.51) mm, rotated rx -11.83 ry -17.7 rz 126.62 deg; joints [5.237, -27.199, 114.574, 232.118, 72.685, -39.907, 143.741]
  MoveL 2378 to (13.81, -56.68, -266.73) mm, rotated rx -11.83 ry -17.7 rz 126.62 deg; joints [5.234, -27.186, 114.574, 232.113, 72.692, -39.898, 143.741]
  MoveL 2379 to (13.64, -56.88, -266.84) mm, rotated rx -11.83 ry -17.7 rz 126.62 deg; joints [5.238, -27.17, 114.552, 232.118, 72.689, -39.902, 143.741]
  MoveL 2380 to (13.4, -57.26, -266.87) mm, rotated rx -11.83 ry -17.7 rz 126.62 deg; joints [5.245, -27.15, 114.516, 232.129, 72.679, -39.916, 143.741]
  MoveL 2381 to (13.16, -57.68, -266.9) mm, rotated rx -11.83 ry -17.7 rz 126.62 deg; joints [5.251, -27.13, 114.476, 232.14, 72.668, -39.932, 143.741]
  MoveL 2382 to (12.96, -58.06, -266.95) mm, rotated rx -11.83 ry -17.7 rz 126.62 deg; joints [5.256, -27.11, 114.441, 232.15, 72.658, -39.946, 143.741]
  MoveL 2383 to (12.76, -58.41, -267.01) mm, rotated rx -11.83 ry -17.7 rz 126.62 deg; joints [5.261, -27.09, 114.407, 232.158, 72.649, -39.957, 143.741]
  MoveL 2384 to (12.56, -58.77, -267.07) mm, rotated rx -11.83 ry -17.7 rz 126.62 deg; joints [5.266, -27.071, 114.373, 232.166, 72.641, -39.969, 143.741]
  MoveL 2385 to (12.35, -59.16, -267.11) mm, rotated rx -11.83 ry -17.7 rz 126.62 deg; joints [5.271, -27.051, 114.336, 232.176, 72.63, -39.984, 143.741]
  MoveL 2386 to (12.12, -59.63, -267.13) mm, rotated rx -11.83 ry -17.7 rz 126.62 deg; joints [5.277, -27.03, 114.292, 232.187, 72.617, -40.002, 143.741]
  MoveL 2387 to (11.87, -60.1, -267.2) mm, rotated rx -11.83 ry -17.7 rz 126.62 deg; joints [5.283, -27.005, 114.248, 232.198, 72.605, -40.019, 143.741]
  MoveL 2388 to (11.63, -60.56, -267.23) mm, rotated rx -11.83 ry -17.7 rz 126.62 deg; joints [5.289, -26.983, 114.204, 232.209, 72.592, -40.037, 143.741]
  MoveL 2389 to (11.41, -61.03, -267.23) mm, rotated rx -11.83 ry -17.7 rz 126.62 deg; joints [5.295, -26.963, 114.161, 232.221, 72.578, -40.056, 143.741]
  MoveL 2390 to (11.18, -61.5, -267.23) mm, rotated rx -11.83 ry -17.7 rz 126.62 deg; joints [5.301, -26.942, 114.117, 232.232, 72.564, -40.076, 143.741]
  MoveL 2391 to (10.91, -62.13, -267.2) mm, rotated rx -11.83 ry -17.7 rz 126.62 deg; joints [5.308, -26.918, 114.059, 232.248, 72.544, -40.104, 143.741]
  MoveL 2392 to (10.64, -62.74, -267.17) mm, rotated rx -11.83 ry -17.7 rz 126.62 deg; joints [5.315, -26.894, 114.004, 232.263, 72.525, -40.13, 143.741]
  MoveL 2393 to (10.39, -63.29, -267.16) mm, rotated rx -11.83 ry -17.7 rz 126.62 deg; joints [5.321, -26.871, 113.954, 232.276, 72.508, -40.153, 143.741]
  MoveL 2394 to (10.17, -63.7, -267.2) mm, rotated rx -11.83 ry -17.7 rz 126.62 deg; joints [5.327, -26.85, 113.914, 232.286, 72.497, -40.168, 143.741]
  MoveL 2395 to (9.97, -64.06, -267.26) mm, rotated rx -11.83 ry -17.7 rz 126.62 deg; joints [5.332, -26.831, 113.88, 232.295, 72.488, -40.181, 143.741]
  MoveL 2396 to (9.77, -64.42, -267.32) mm, rotated rx -11.83 ry -17.7 rz 126.62 deg; joints [5.336, -26.811, 113.846, 232.304, 72.479, -40.194, 143.741]
  MoveL 2397 to (9.56, -64.81, -267.35) mm, rotated rx -11.83 ry -17.7 rz 126.62 deg; joints [5.341, -26.792, 113.809, 232.313, 72.469, -40.208, 143.741]
  MoveL 2398 to (8.9, -66.23, -267.35) mm, rotated rx -11.83 ry -17.7 rz 126.62 deg; joints [5.358, -26.731, 113.677, 232.348, 72.426, -40.268, 143.741]
  MoveL 2399 to (7.47, -68.75, -267.73) mm, rotated rx -11.83 ry -17.7 rz 126.62 deg; joints [5.394, -26.595, 113.435, 232.41, 72.363, -40.357, 143.741]
  MoveL 2400 to (6.69, -69.73, -268.2) mm, rotated rx -11.83 ry -17.7 rz 126.62 deg; joints [5.412, -26.519, 113.334, 232.435, 72.349, -40.378, 143.741]
  MoveL 2401 to (5.88, -70.53, -268.86) mm, rotated rx -11.83 ry -17.7 rz 126.62 deg; joints [5.431, -26.436, 113.244, 232.456, 72.346, -40.384, 143.741]
  MoveL 2402 to (5.02, -71.15, -269.71) mm, rotated rx -11.83 ry -17.7 rz 126.62 deg; joints [5.45, -26.348, 113.168, 232.472, 72.354, -40.375, 143.741]
  MoveL 2403 to (4.12, -71.59, -270.74) mm, rotated rx -11.83 ry -17.7 rz 126.62 deg; joints [5.47, -26.253, 113.104, 232.484, 72.373, -40.351, 143.741]
  MoveL 2404 to (2.2, -71.93, -273.38) mm, rotated rx -11.83 ry -17.7 rz 126.62 deg; joints [5.511, -26.047, 113.013, 232.497, 72.445, -40.256, 143.741]
  MoveL 2405 to (0.66, -71.56, -276.02) mm, rotated rx -11.83 ry -17.7 rz 126.62 deg; joints [5.542, -25.872, 112.988, 232.49, 72.538, -40.132, 143.741]
  MoveL 2406 to (0.22, -71.13, -277.05) mm, rotated rx -11.83 ry -17.7 rz 126.62 deg; joints [5.549, -25.816, 113.006, 232.479, 72.583, -40.071, 143.741]
  MoveL 2407 to (0.02, -70.52, -277.9) mm, rotated rx -11.83 ry -17.7 rz 126.62 deg; joints [5.551, -25.782, 113.044, 232.463, 72.627, -40.011, 143.741]
  MoveL 2408 to (0.04, -69.75, -278.56) mm, rotated rx -11.83 ry -17.7 rz 126.62 deg; joints [5.547, -25.769, 113.103, 232.441, 72.67, -39.952, 143.741]
  MoveL 2409 to (0.29, -68.81, -279.03) mm, rotated rx -11.83 ry -17.7 rz 126.62 deg; joints [5.537, -25.778, 113.182, 232.415, 72.713, -39.893, 143.741]
  MoveL 2410 to (0.76, -67.7, -279.31) mm, rotated rx -11.83 ry -17.7 rz 126.62 deg; joints [5.522, -25.807, 113.281, 232.382, 72.755, -39.835, 143.741]
  MoveL 2411 to (1.47, -66.42, -279.41) mm, rotated rx -11.83 ry -17.7 rz 126.62 deg; joints [5.502, -25.859, 113.401, 232.345, 72.796, -39.778, 143.741]
  MoveL 2412 to (1.74, -65.97, -279.41) mm, rotated rx -11.83 ry -17.7 rz 126.62 deg; joints [5.494, -25.879, 113.444, 232.331, 72.809, -39.759, 143.741]
  MoveL 2413 to (1.98, -65.58, -279.39) mm, rotated rx -11.83 ry -17.7 rz 126.62 deg; joints [5.487, -25.899, 113.482, 232.32, 72.82, -39.743, 143.741]
  MoveL 2414 to (2.21, -65.25, -279.34) mm, rotated rx -11.83 ry -17.7 rz 126.62 deg; joints [5.48, -25.917, 113.514, 232.31, 72.829, -39.731, 143.741]
  MoveL 2415 to (2.44, -64.93, -279.28) mm, rotated rx -11.83 ry -17.7 rz 126.62 deg; joints [5.474, -25.936, 113.546, 232.3, 72.837, -39.72, 143.741]
  MoveL 2416 to (2.68, -64.57, -279.24) mm, rotated rx -11.83 ry -17.7 rz 126.62 deg; joints [5.468, -25.955, 113.581, 232.29, 72.846, -39.707, 143.741]
  MoveL 2417 to (2.94, -64.16, -279.21) mm, rotated rx -11.83 ry -17.7 rz 126.62 deg; joints [5.46, -25.976, 113.621, 232.277, 72.858, -39.691, 143.741]
  MoveL 2418 to (3.21, -63.71, -279.21) mm, rotated rx -11.83 ry -17.7 rz 126.62 deg; joints [5.452, -25.996, 113.664, 232.264, 72.871, -39.672, 143.741]
  MoveL 2419 to (3.46, -63.31, -279.19) mm, rotated rx -11.83 ry -17.7 rz 126.62 deg; joints [5.445, -26.016, 113.702, 232.253, 72.882, -39.656, 143.741]
  MoveL 2420 to (3.68, -62.97, -279.14) mm, rotated rx -11.83 ry -17.7 rz 126.62 deg; joints [5.439, -26.034, 113.735, 232.243, 72.891, -39.645, 143.741]
  MoveL 2421 to (3.9, -62.65, -279.08) mm, rotated rx -11.83 ry -17.7 rz 126.62 deg; joints [5.434, -26.053, 113.767, 232.234, 72.899, -39.634, 143.741]
  MoveL 2422 to (4.14, -62.29, -279.03) mm, rotated rx -11.83 ry -17.7 rz 126.62 deg; joints [5.427, -26.073, 113.802, 232.224, 72.908, -39.62, 143.741]
  MoveL 2423 to (4.4, -61.87, -279.01) mm, rotated rx -11.83 ry -17.7 rz 126.62 deg; joints [5.42, -26.093, 113.842, 232.212, 72.92, -39.604, 143.741]
  MoveL 2424 to (4.66, -61.42, -279.01) mm, rotated rx -11.83 ry -17.7 rz 126.62 deg; joints [5.412, -26.114, 113.885, 232.199, 72.933, -39.585, 143.741]
  MoveL 2425 to (5.24, -60.61, -278.99) mm, rotated rx -11.83 ry -17.7 rz 126.62 deg; joints [5.395, -26.153, 113.963, 232.172, 72.956, -39.553, 143.741]
  MoveC 2426 to (6.06, -59.51, -278.99) mm, rotated rx -11.83 ry -17.7 rz 126.62 deg; joints [5.369, -26.208, 114.071, 232.132, 72.989, -39.508, 143.741] to (6.74, -58.31, -278.99) mm, rotated rx -11.83 ry -17.7 rz 126.62 deg; joints [5.349, -26.261, 114.184, 232.098, 73.025, -39.458, 143.741]
  MoveL 2427 to (6.74, -58.31, -278.98) mm, rotated rx -11.83 ry -17.7 rz 126.62 deg; joints [5.349, -26.261, 114.184, 232.099, 73.024, -39.459, 143.741]
  MoveL 2428 to (7.12, -57.77, -278.96) mm, rotated rx -11.83 ry -17.7 rz 126.62 deg; joints [5.338, -26.288, 114.237, 232.081, 73.04, -39.437, 143.741]
  MoveL 2429 to (7.49, -57.33, -278.94) mm, rotated rx -11.83 ry -17.7 rz 126.62 deg; joints [5.326, -26.312, 114.281, 232.064, 73.052, -39.421, 143.741]
  MoveL 2430 to (7.74, -57.15, -278.84) mm, rotated rx -11.83 ry -17.7 rz 126.62 deg; joints [5.319, -26.329, 114.301, 232.056, 73.054, -39.417, 143.741]
  MoveL 2431 to (7.73, -57.21, -278.64) mm, rotated rx -11.83 ry -17.7 rz 126.62 deg; joints [5.321, -26.339, 114.298, 232.061, 73.046, -39.428, 143.741]
  MoveL 2432 to (7.45, -57.53, -278.33) mm, rotated rx -11.83 ry -17.7 rz 126.62 deg; joints [5.334, -26.34, 114.269, 232.082, 73.028, -39.453, 143.741]
  MoveL 2433 to (7.55, -57.9, -277.71) mm, rotated rx -11.83 ry -17.7 rz 126.62 deg; joints [5.336, -26.366, 114.247, 232.095, 72.998, -39.494, 143.741]
  MoveL 2434 to (9.35, -56.94, -277.7) mm, rotated rx -11.83 ry -17.7 rz 126.62 deg; joints [5.268, -26.44, 114.36, 232.018, 73.02, -39.459, 143.741]
  MoveL 2435 to (11.27, -56, -277.65) mm, rotated rx -11.83 ry -17.7 rz 126.62 deg; joints [5.196, -26.519, 114.475, 231.936, 73.04, -39.428, 143.741]
  MoveL 2436 to (13.34, -55.05, -277.52) mm, rotated rx -11.83 ry -17.7 rz 126.62 deg; joints [5.118, -26.606, 114.593, 231.85, 73.058, -39.4, 143.741]
  MoveL 2437 to (15.36, -54.11, -277.42) mm, rotated rx -11.83 ry -17.7 rz 126.62 deg; joints [5.042, -26.689, 114.709, 231.766, 73.076, -39.372, 143.741]
  MoveL 2438 to (17.32, -53.21, -277.25) mm, rotated rx -11.83 ry -17.7 rz 126.62 deg; joints [4.969, -26.775, 114.821, 231.686, 73.09, -39.348, 143.741]
  MoveL 2439 to (19.09, -52.4, -277.1) mm, rotated rx -11.83 ry -17.7 rz 126.62 deg; joints [4.902, -26.851, 114.922, 231.614, 73.104, -39.326, 143.741]
  MoveL 2440 to (20.96, -51.52, -277.05) mm, rotated rx -11.83 ry -17.7 rz 126.62 deg; joints [4.831, -26.926, 115.029, 231.534, 73.122, -39.299, 143.741]
  MoveL 2441 to (22.92, -50.61, -276.98) mm, rotated rx -11.83 ry -17.7 rz 126.62 deg; joints [4.756, -27.006, 115.14, 231.452, 73.139, -39.272, 143.741]
  MoveL 2442 to (25.05, -49.62, -276.83) mm, rotated rx -11.83 ry -17.7 rz 126.62 deg; joints [4.676, -27.097, 115.262, 231.363, 73.156, -39.245, 143.741]
  MoveL 2443 to (26.75, -48.82, -276.71) mm, rotated rx -11.83 ry -17.7 rz 126.62 deg; joints [4.611, -27.169, 115.359, 231.293, 73.17, -39.223, 143.741]
  MoveL 2444 to (28.91, -47.81, -276.5) mm, rotated rx -11.83 ry -17.7 rz 126.62 deg; joints [4.531, -27.265, 115.483, 231.205, 73.186, -39.199, 143.741]
  MoveL 2445 to (30.61, -47.01, -276.39) mm, rotated rx -11.83 ry -17.7 rz 126.62 deg; joints [4.466, -27.337, 115.58, 231.134, 73.2, -39.178, 143.741]
  MoveL 2446 to (32.54, -46.09, -276.22) mm, rotated rx -11.83 ry -17.7 rz 126.62 deg; joints [4.393, -27.421, 115.69, 231.055, 73.215, -39.155, 143.741]
  MoveL 2447 to (34.7, -45.07, -276.17) mm, rotated rx -11.83 ry -17.7 rz 126.62 deg; joints [4.31, -27.508, 115.812, 230.963, 73.235, -39.124, 143.741]
  MoveL 2448 to (36.4, -44.27, -276.06) mm, rotated rx -11.83 ry -17.7 rz 126.62 deg; joints [4.245, -27.58, 115.909, 230.892, 73.249, -39.104, 143.741]
  MoveL 2449 to (38.32, -43.34, -275.9) mm, rotated rx -11.83 ry -17.7 rz 126.62 deg; joints [4.173, -27.665, 116.019, 230.813, 73.263, -39.081, 143.741]
  MoveL 2450 to (40.48, -42.32, -275.85) mm, rotated rx -11.83 ry -17.7 rz 126.62 deg; joints [4.089, -27.751, 116.14, 230.721, 73.284, -39.052, 143.741]
  MoveL 2451 to (42.17, -41.51, -275.74) mm, rotated rx -11.83 ry -17.7 rz 126.62 deg; joints [4.024, -27.823, 116.236, 230.65, 73.297, -39.031, 143.741]
  MoveL 2452 to (44.18, -40.55, -275.63) mm, rotated rx -11.83 ry -17.7 rz 126.62 deg; joints [3.947, -27.907, 116.35, 230.566, 73.314, -39.006, 143.741]
  MoveL 2453 to (46.19, -39.59, -275.56) mm, rotated rx -11.83 ry -17.7 rz 126.62 deg; joints [3.869, -27.989, 116.463, 230.48, 73.332, -38.979, 143.741]
  MoveL 2454 to (47.87, -38.75, -275.38) mm, rotated rx -11.83 ry -17.7 rz 126.62 deg; joints [3.806, -28.066, 116.561, 230.412, 73.345, -38.961, 143.741]
  MoveL 2455 to (49.41, -37.95, -275.13) mm, rotated rx -11.83 ry -17.7 rz 126.62 deg; joints [3.749, -28.143, 116.654, 230.351, 73.354, -38.947, 143.741]
  MoveL 2456 to (50.83, -37.18, -274.78) mm, rotated rx -11.83 ry -17.7 rz 126.62 deg; joints [3.698, -28.221, 116.745, 230.297, 73.361, -38.936, 143.741]
  MoveL 2457 to (49.35, -37.42, -274.09) mm, rotated rx -11.83 ry -17.7 rz 126.62 deg; joints [3.77, -28.219, 116.708, 230.377, 73.341, -38.965, 143.741]
  MoveL 2458 to (49.57, -37.36, -274.08) mm, rotated rx -11.83 ry -17.7 rz 126.62 deg; joints [3.761, -28.226, 116.717, 230.368, 73.341, -38.964, 143.741]
  MoveL 2459 to (49.87, -37.32, -274.07) mm, rotated rx -11.83 ry -17.7 rz 126.62 deg; joints [3.749, -28.235, 116.725, 230.356, 73.34, -38.964, 143.741]
  MoveL 2460 to (50.32, -37.33, -274.04) mm, rotated rx -11.83 ry -17.7 rz 126.62 deg; joints [3.73, -28.248, 116.731, 230.338, 73.336, -38.969, 143.741]
  MoveL 2461 to (50.86, -37.37, -274) mm, rotated rx -11.83 ry -17.7 rz 126.62 deg; joints [3.707, -28.262, 116.737, 230.317, 73.33, -38.975, 143.741]
  MoveL 2462 to (51.47, -37.44, -273.96) mm, rotated rx -11.83 ry -17.7 rz 126.62 deg; joints [3.681, -28.277, 116.742, 230.294, 73.323, -38.983, 143.741]
  MoveL 2463 to (54.06, -37.83, -273.96) mm, rotated rx -11.83 ry -17.7 rz 126.62 deg; joints [3.569, -28.328, 116.75, 230.191, 73.293, -39.015, 143.741]
  MoveL 2464 to (54.66, -37.9, -273.93) mm, rotated rx -11.83 ry -17.7 rz 126.62 deg; joints [3.543, -28.342, 116.753, 230.167, 73.286, -39.023, 143.741]
  MoveL 2465 to (55.35, -37.98, -273.87) mm, rotated rx -11.83 ry -17.7 rz 126.62 deg; joints [3.514, -28.359, 116.759, 230.141, 73.278, -39.033, 143.741]
  MoveL 2466 to (55.97, -38.05, -273.84) mm, rotated rx -11.83 ry -17.7 rz 126.62 deg; joints [3.488, -28.374, 116.762, 230.117, 73.27, -39.041, 143.741]
  MoveL 2467 to (56.49, -38.13, -273.84) mm, rotated rx -11.83 ry -17.7 rz 126.62 deg; joints [3.465, -28.384, 116.764, 230.097, 73.264, -39.047, 143.741]
  MoveL 2468 to (56.97, -38.2, -273.83) mm, rotated rx -11.83 ry -17.7 rz 126.62 deg; joints [3.444, -28.394, 116.765, 230.077, 73.258, -39.054, 143.741]
  MoveL 2469 to (57.49, -38.28, -273.83) mm, rotated rx -11.83 ry -17.7 rz 126.62 deg; joints [3.422, -28.404, 116.767, 230.057, 73.252, -39.06, 143.741]
  MoveL 2470 to (58, -38.36, -273.83) mm, rotated rx -11.83 ry -17.7 rz 126.62 deg; joints [3.4, -28.414, 116.768, 230.037, 73.246, -39.067, 143.741]
  MoveL 2471 to (58.48, -38.42, -273.8) mm, rotated rx -11.83 ry -17.7 rz 126.62 deg; joints [3.379, -28.426, 116.771, 230.018, 73.24, -39.073, 143.741]
  MoveL 2472 to (58.94, -38.47, -273.75) mm, rotated rx -11.83 ry -17.7 rz 126.62 deg; joints [3.36, -28.438, 116.774, 230.001, 73.234, -39.08, 143.741]
  MoveL 2473 to (59.43, -38.54, -273.73) mm, rotated rx -11.83 ry -17.7 rz 126.62 deg; joints [3.339, -28.449, 116.777, 229.982, 73.228, -39.087, 143.741]
  MoveL 2474 to (59.96, -38.62, -273.73) mm, rotated rx -11.83 ry -17.7 rz 126.62 deg; joints [3.317, -28.459, 116.778, 229.961, 73.222, -39.093, 143.741]
  MoveL 2475 to (60.99, -38.77, -273.73) mm, rotated rx -11.83 ry -17.7 rz 126.62 deg; joints [3.272, -28.48, 116.781, 229.92, 73.209, -39.106, 143.741]
  Set speed (1000.0 mm/s)
  MoveL 2476 to (80.59, -47.91, -273.73) mm, rotated rx -11.83 ry -17.7 rz 126.62 deg; joints [2.389, -28.666, 116.307, 229.186, 72.757, -39.611, 143.741]
  Print: /'Flow1'
  Set speed (1000.0 mm/s)
  MoveL 2477 to (43.45, 100.59, -76.32) mm, rotated rx 164.15 ry 19.7 rz -117.91 deg; joints [7.261, -26.764, 91.379, 208.398, 85.726, 6.48, 26.033]
  Set speed (1000.0 mm/s)
  MoveL 2478 to (6.14, 75.62, -69.16) mm, rotated rx -152.51 ry -6.42 rz -112.51 deg; joints [12.894, -19.518, 66.565, 214.587, 99.097, 37.073, 26.033]
  Set speed (100.0 mm/s)
  MoveL 2479 to (-53.46, 33.88, -69.16) mm, rotated rx -152.51 ry -6.42 rz -112.51 deg; joints [15.009, -20.083, 69.393, 216.193, 101.757, 37.236, 26.033]
  MoveL 2480 to (-53.98, 33.91, -69.16) mm, rotated rx -152.51 ry -6.42 rz -112.51 deg; joints [15.025, -20.086, 69.388, 216.203, 101.757, 37.223, 26.033]
  MoveL 2481 to (-54.63, 33.89, -69.07) mm, rotated rx -152.51 ry -6.42 rz -112.51 deg; joints [15.045, -20.083, 69.374, 216.215, 101.757, 37.206, 26.033]
  MoveL 2482 to (-55.22, 33.89, -69.01) mm, rotated rx -152.51 ry -6.42 rz -112.51 deg; joints [15.064, -20.082, 69.365, 216.226, 101.757, 37.19, 26.033]
  MoveL 2483 to (-55.79, 33.91, -68.99) mm, rotated rx -152.51 ry -6.42 rz -112.51 deg; joints [15.081, -20.084, 69.357, 216.236, 101.756, 37.176, 26.033]
  MoveL 2484 to (-59.45, 34.11, -68.99) mm, rotated rx -152.51 ry -6.42 rz -112.51 deg; joints [15.194, -20.106, 69.323, 216.302, 101.754, 37.081, 26.033]
  MoveL 2485 to (-60.89, 34.25, -69.08) mm, rotated rx -152.51 ry -6.42 rz -112.51 deg; joints [15.237, -20.121, 69.315, 216.327, 101.752, 37.043, 26.033]
  MoveL 2486 to (-62.05, 34.49, -69.34) mm, rotated rx -152.51 ry -6.42 rz -112.51 deg; joints [15.271, -20.149, 69.322, 216.347, 101.749, 37.013, 26.033]
  MoveL 2487 to (-62.93, 34.84, -69.79) mm, rotated rx -152.51 ry -6.42 rz -112.51 deg; joints [15.295, -20.188, 69.345, 216.36, 101.745, 36.99, 26.033]
  MoveL 2488 to (-63.27, 35.06, -70.08) mm, rotated rx -152.51 ry -6.42 rz -112.51 deg; joints [15.303, -20.212, 69.362, 216.364, 101.742, 36.982, 26.033]
  MoveL 2489 to (-63.53, 35.3, -70.41) mm, rotated rx -152.51 ry -6.42 rz -112.51 deg; joints [15.309, -20.239, 69.383, 216.367, 101.74, 36.975, 26.033]
  MoveL 2490 to (-63.84, 35.86, -71.21) mm, rotated rx -152.51 ry -6.42 rz -112.51 deg; joints [15.312, -20.303, 69.437, 216.368, 101.733, 36.967, 26.033]
  MoveL 2491 to (-63.88, 36.53, -72.18) mm, rotated rx -152.51 ry -6.42 rz -112.51 deg; joints [15.306, -20.378, 69.505, 216.364, 101.725, 36.966, 26.033]
  MoveL 2492 to (-63.1, 38.19, -74.67) mm, rotated rx -152.51 ry -6.42 rz -112.51 deg; joints [15.264, -20.564, 69.688, 216.336, 101.706, 36.987, 26.033]
  MoveL 2493 to (-61.53, 39.75, -77.15) mm, rotated rx -152.51 ry -6.42 rz -112.51 deg; joints [15.198, -20.745, 69.88, 216.295, 101.689, 37.029, 26.033]
  MoveL 2494 to (-59.51, 40.72, -78.93) mm, rotated rx -152.51 ry -6.42 rz -112.51 deg; joints [15.124, -20.869, 70.033, 216.25, 101.684, 37.086, 26.033]
  MoveL 2495 to (-58.34, 40.98, -79.55) mm, rotated rx -152.51 ry -6.42 rz -112.51 deg; joints [15.084, -20.91, 70.094, 216.227, 101.685, 37.12, 26.033]
  MoveL 2496 to (-57.05, 41.08, -79.99) mm, rotated rx -152.51 ry -6.42 rz -112.51 deg; joints [15.042, -20.936, 70.146, 216.203, 101.689, 37.158, 26.033]
  MoveL 2497 to (-54.14, 40.85, -80.35) mm, rotated rx -152.51 ry -6.42 rz -112.51 deg; joints [14.952, -20.946, 70.22, 216.152, 101.707, 37.245, 26.033]
  MoveL 2498 to (-51.04, 40.32, -80.35) mm, rotated rx -152.51 ry -6.42 rz -112.51 deg; joints [14.859, -20.928, 70.274, 216.101, 101.729, 37.339, 26.033]
  MoveL 2499 to (-50.56, 40.25, -80.37) mm, rotated rx -152.51 ry -6.42 rz -112.51 deg; joints [14.844, -20.926, 70.283, 216.092, 101.733, 37.353, 26.033]
  MoveL 2500 to (-50.1, 40.2, -80.41) mm, rotated rx -152.51 ry -6.42 rz -112.51 deg; joints [14.83, -20.926, 70.294, 216.085, 101.736, 37.367, 26.033]
  MoveL 2501 to (-49.68, 40.17, -80.47) mm, rotated rx -152.51 ry -6.42 rz -112.51 deg; joints [14.818, -20.929, 70.305, 216.077, 101.738, 37.379, 26.033]
  MoveL 2502 to (-49.24, 40.13, -80.52) mm, rotated rx -152.51 ry -6.42 rz -112.51 deg; joints [14.804, -20.93, 70.316, 216.07, 101.741, 37.393, 26.033]
  MoveL 2503 to (-48.7, 40.05, -80.55) mm, rotated rx -152.51 ry -6.42 rz -112.51 deg; joints [14.788, -20.928, 70.327, 216.061, 101.745, 37.409, 26.033]
  MoveL 2504 to (-48.06, 39.96, -80.59) mm, rotated rx -152.51 ry -6.42 rz -112.51 deg; joints [14.768, -20.927, 70.341, 216.05, 101.749, 37.428, 26.033]
  MoveL 2505 to (-47.5, 39.9, -80.65) mm, rotated rx -152.51 ry -6.42 rz -112.51 deg; joints [14.751, -20.928, 70.355, 216.04, 101.753, 37.445, 26.033]
  MoveL 2506 to (-47.05, 39.87, -80.72) mm, rotated rx -152.51 ry -6.42 rz -112.51 deg; joints [14.737, -20.931, 70.368, 216.032, 101.756, 37.459, 26.033]
  MoveL 2507 to (-46.62, 39.82, -80.77) mm, rotated rx -152.51 ry -6.42 rz -112.51 deg; joints [14.724, -20.932, 70.379, 216.025, 101.759, 37.472, 26.033]
  MoveL 2508 to (-46.15, 39.76, -80.79) mm, rotated rx -152.51 ry -6.42 rz -112.51 deg; joints [14.709, -20.931, 70.388, 216.017, 101.762, 37.486, 26.033]
  MoveL 2509 to (-45.63, 39.67, -80.79) mm, rotated rx -152.51 ry -6.42 rz -112.51 deg; joints [14.694, -20.927, 70.397, 216.008, 101.766, 37.502, 26.033]
  MoveL 2510 to (-45.1, 39.58, -80.79) mm, rotated rx -152.51 ry -6.42 rz -112.51 deg; joints [14.678, -20.924, 70.406, 215.999, 101.77, 37.518, 26.033]
  MoveL 2511 to (-44.53, 39.49, -80.8) mm, rotated rx -152.51 ry -6.42 rz -112.51 deg; joints [14.661, -20.921, 70.416, 215.99, 101.773, 37.534, 26.033]
  MoveL 2512 to (-43.88, 39.42, -80.84) mm, rotated rx -152.51 ry -6.42 rz -112.51 deg; joints [14.64, -20.92, 70.428, 215.978, 101.777, 37.554, 26.033]
  MoveL 2513 to (-43.28, 39.38, -80.9) mm, rotated rx -152.51 ry -6.42 rz -112.51 deg; joints [14.622, -20.921, 70.441, 215.968, 101.779, 37.571, 26.033]
  MoveL 2514 to (-42.83, 39.38, -81.01) mm, rotated rx -152.51 ry -6.42 rz -112.51 deg; joints [14.608, -20.926, 70.455, 215.96, 101.781, 37.584, 26.033]
  MoveL 2515 to (-42.83, 39.37, -81.24) mm, rotated rx -152.51 ry -6.42 rz -112.51 deg; joints [14.607, -20.944, 70.484, 215.96, 101.789, 37.59, 26.033]
  MoveL 2516 to (-43.22, 39.31, -81.6) mm, rotated rx -152.51 ry -6.42 rz -112.51 deg; joints [14.619, -20.974, 70.527, 215.97, 101.805, 37.592, 26.033]
  MoveL 2517 to (-43.83, 39.9, -82.56) mm, rotated rx -152.51 ry -6.42 rz -112.51 deg; joints [14.631, -21.052, 70.595, 215.977, 101.802, 37.58, 26.033]
  MoveL 2518 to (-41.89, 40.77, -82.56) mm, rotated rx -152.51 ry -6.42 rz -112.51 deg; joints [14.564, -21.038, 70.544, 215.929, 101.746, 37.593, 26.033]
  MoveL 2519 to (-39.81, 41.74, -82.69) mm, rotated rx -152.51 ry -6.42 rz -112.51 deg; joints [14.492, -21.032, 70.501, 215.877, 101.688, 37.609, 26.033]
  MoveL 2520 to (-37.82, 42.64, -82.75) mm, rotated rx -152.51 ry -6.42 rz -112.51 deg; joints [14.424, -21.022, 70.454, 215.828, 101.632, 37.624, 26.033]
  MoveL 2521 to (-35.9, 43.53, -82.88) mm, rotated rx -152.51 ry -6.42 rz -112.51 deg; joints [14.358, -21.017, 70.415, 215.781, 101.58, 37.64, 26.033]
  MoveL 2522 to (-33.95, 44.42, -83.04) mm, rotated rx -152.51 ry -6.42 rz -112.51 deg; joints [14.291, -21.015, 70.379, 215.733, 101.527, 37.656, 26.033]
  MoveL 2523 to (-32.02, 45.3, -83.16) mm, rotated rx -152.51 ry -6.42 rz -112.51 deg; joints [14.224, -21.009, 70.339, 215.686, 101.474, 37.671, 26.033]
  MoveL 2524 to (-30.07, 46.2, -83.37) mm, rotated rx -152.51 ry -6.42 rz -112.51 deg; joints [14.157, -21.01, 70.308, 215.638, 101.422, 37.689, 26.033]
  MoveL 2525 to (-28.13, 47.07, -83.48) mm, rotated rx -152.51 ry -6.42 rz -112.51 deg; joints [14.09, -21.004, 70.267, 215.591, 101.369, 37.704, 26.033]
  MoveL 2526 to (-26.18, 47.95, -83.54) mm, rotated rx -152.51 ry -6.42 rz -112.51 deg; joints [14.023, -20.992, 70.219, 215.543, 101.313, 37.718, 26.033]
  MoveL 2527 to (-24.21, 48.84, -83.68) mm, rotated rx -152.51 ry -6.42 rz -112.51 deg; joints [13.956, -20.988, 70.18, 215.495, 101.26, 37.735, 26.033]
  MoveL 2528 to (-22.18, 49.75, -83.86) mm, rotated rx -152.51 ry -6.42 rz -112.51 deg; joints [13.886, -20.985, 70.143, 215.445, 101.205, 37.753, 26.033]
  MoveL 2529 to (-20.15, 50.66, -84.04) mm, rotated rx -152.51 ry -6.42 rz -112.51 deg; joints [13.816, -20.982, 70.106, 215.396, 101.151, 37.771, 26.033]
  MoveL 2530 to (-18.43, 51.42, -84.29) mm, rotated rx -152.51 ry -6.42 rz -112.51 deg; joints [13.757, -20.987, 70.086, 215.355, 101.109, 37.788, 26.033]
  MoveL 2531 to (-16, 52.51, -84.39) mm, rotated rx -152.51 ry -6.42 rz -112.51 deg; joints [13.673, -20.974, 70.028, 215.295, 101.04, 37.807, 26.033]
  Set speed (1000.0 mm/s)
  MoveL 2532 to (21.11, 78.49, -84.39) mm, rotated rx -152.51 ry -6.42 rz -112.51 deg; joints [12.359, -20.589, 68.193, 214.294, 99.351, 37.695, 26.033]
  Set speed (1000.0 mm/s)
  MoveL 2533 to (24.4, 73.79, -96.27) mm, rotated rx -152.51 ry -6.42 rz -112.51 deg; joints [12.24, -21.505, 69.929, 214.295, 99.984, 38.231, 26.033]
  Set speed (100.0 mm/s)
  MoveL 2534 to (0.9, 57.34, -96.27) mm, rotated rx -152.51 ry -6.42 rz -112.51 deg; joints [13.075, -21.747, 71.092, 214.937, 101.053, 38.303, 26.033]
  MoveL 2535 to (-0.74, 56.86, -96.03) mm, rotated rx -152.51 ry -6.42 rz -112.51 deg; joints [13.13, -21.742, 71.095, 214.974, 101.08, 38.277, 26.033]
  MoveL 2536 to (-2.68, 56.26, -95.96) mm, rotated rx -152.51 ry -6.42 rz -112.51 deg; joints [13.195, -21.754, 71.126, 215.019, 101.12, 38.254, 26.033]
  MoveL 2537 to (-4.64, 55.66, -95.82) mm, rotated rx -152.51 ry -6.42 rz -112.51 deg; joints [13.26, -21.76, 71.149, 215.064, 101.158, 38.228, 26.033]
  MoveL 2538 to (-7, 54.95, -95.68) mm, rotated rx -152.51 ry -6.42 rz -112.51 deg; joints [13.339, -21.769, 71.178, 215.118, 101.204, 38.197, 26.033]
  MoveL 2539 to (-9.03, 54.32, -95.68) mm, rotated rx -152.51 ry -6.42 rz -112.51 deg; joints [13.407, -21.786, 71.219, 215.165, 101.249, 38.174, 26.033]
  MoveL 2540 to (-11.29, 53.61, -95.53) mm, rotated rx -152.51 ry -6.42 rz -112.51 deg; joints [13.483, -21.793, 71.245, 215.216, 101.293, 38.145, 26.033]
  MoveL 2541 to (-13.19, 53.03, -95.34) mm, rotated rx -152.51 ry -6.42 rz -112.51 deg; joints [13.547, -21.795, 71.26, 215.26, 101.328, 38.118, 26.033]
  MoveL 2542 to (-15.15, 52.43, -95.25) mm, rotated rx -152.51 ry -6.42 rz -112.51 deg; joints [13.612, -21.803, 71.287, 215.305, 101.368, 38.093, 26.033]
  MoveL 2543 to (-17.19, 51.79, -95.03) mm, rotated rx -152.51 ry -6.42 rz -112.51 deg; joints [13.681, -21.803, 71.301, 215.351, 101.405, 38.064, 26.033]
  MoveL 2544 to (-19.2, 51.15, -94.87) mm, rotated rx -152.51 ry -6.42 rz -112.51 deg; joints [13.749, -21.807, 71.322, 215.397, 101.444, 38.038, 26.033]
  MoveL 2545 to (-21.22, 50.52, -94.76) mm, rotated rx -152.51 ry -6.42 rz -112.51 deg; joints [13.816, -21.815, 71.348, 215.444, 101.485, 38.012, 26.033]
  MoveL 2546 to (-23.26, 49.87, -94.6) mm, rotated rx -152.51 ry -6.42 rz -112.51 deg; joints [13.885, -21.818, 71.368, 215.491, 101.524, 37.985, 26.033]
  MoveL 2547 to (-25.28, 49.22, -94.45) mm, rotated rx -152.51 ry -6.42 rz -112.51 deg; joints [13.953, -21.823, 71.39, 215.537, 101.564, 37.958, 26.033]
  MoveL 2548 to (-27.36, 48.56, -94.39) mm, rotated rx -152.51 ry -6.42 rz -112.51 deg; joints [14.023, -21.834, 71.421, 215.585, 101.606, 37.933, 26.033]
  MoveL 2549 to (-29.38, 47.9, -94.18) mm, rotated rx -152.51 ry -6.42 rz -112.51 deg; joints [14.091, -21.833, 71.436, 215.632, 101.645, 37.905, 26.033]
  MoveL 2550 to (-31.4, 47.25, -94.05) mm, rotated rx -152.51 ry -6.42 rz -112.51 deg; joints [14.159, -21.839, 71.46, 215.678, 101.685, 37.879, 26.033]
  MoveL 2551 to (-33.46, 46.58, -93.93) mm, rotated rx -152.51 ry -6.42 rz -112.51 deg; joints [14.228, -21.845, 71.484, 215.726, 101.726, 37.853, 26.033]
  MoveL 2552 to (-35.1, 45.91, -93.72) mm, rotated rx -152.51 ry -6.42 rz -112.51 deg; joints [14.285, -21.841, 71.5, 215.765, 101.763, 37.834, 26.033]
  MoveL 2553 to (-36.41, 45.23, -93.37) mm, rotated rx -152.51 ry -6.42 rz -112.51 deg; joints [14.331, -21.824, 71.502, 215.798, 101.796, 37.82, 26.033]
  MoveL 2554 to (-37.38, 44.51, -92.85) mm, rotated rx -152.51 ry -6.42 rz -112.51 deg; joints [14.368, -21.792, 71.487, 215.824, 101.825, 37.812, 26.033]
  MoveL 2555 to (-35.84, 44.51, -91.99) mm, rotated rx -152.51 ry -6.42 rz -112.51 deg; joints [14.323, -21.716, 71.396, 215.792, 101.796, 37.827, 26.033]
  MoveL 2556 to (-36.64, 44.44, -91.99) mm, rotated rx -152.51 ry -6.42 rz -112.51 deg; joints [14.348, -21.721, 71.398, 215.808, 101.802, 37.811, 26.033]
  MoveL 2557 to (-37.34, 44.44, -91.99) mm, rotated rx -152.51 ry -6.42 rz -112.51 deg; joints [14.37, -21.726, 71.395, 215.822, 101.804, 37.795, 26.033]
  MoveL 2558 to (-37.97, 44.54, -91.98) mm, rotated rx -152.51 ry -6.42 rz -112.51 deg; joints [14.389, -21.73, 71.384, 215.832, 101.8, 37.776, 26.033]
  MoveL 2559 to (-38.62, 44.68, -91.96) mm, rotated rx -152.51 ry -6.42 rz -112.51 deg; joints [14.409, -21.733, 71.37, 215.843, 101.793, 37.755, 26.033]
  MoveL 2560 to (-39.36, 44.87, -91.93) mm, rotated rx -152.51 ry -6.42 rz -112.51 deg; joints [14.431, -21.735, 71.35, 215.855, 101.783, 37.73, 26.033]
  MoveL 2561 to (-41.37, 45.47, -91.93) mm, rotated rx -152.51 ry -6.42 rz -112.51 deg; joints [14.49, -21.748, 71.3, 215.885, 101.754, 37.661, 26.033]
  MoveL 2562 to (-41.8, 45.58, -91.91) mm, rotated rx -152.51 ry -6.42 rz -112.51 deg; joints [14.502, -21.749, 71.287, 215.892, 101.748, 37.646, 26.033]
  MoveL 2563 to (-42.81, 45.88, -91.91) mm, rotated rx -152.51 ry -6.42 rz -112.51 deg; joints [14.532, -21.755, 71.262, 215.907, 101.734, 37.611, 26.033]
  MoveL 2564 to (-43.29, 46.02, -91.9) mm, rotated rx -152.51 ry -6.42 rz -112.51 deg; joints [14.546, -21.758, 71.25, 215.915, 101.727, 37.594, 26.033]
  MoveL 2565 to (-43.76, 46.15, -91.89) mm, rotated rx -152.51 ry -6.42 rz -112.51 deg; joints [14.56, -21.76, 71.237, 215.922, 101.72, 37.578, 26.033]
  MoveL 2566 to (-44.23, 46.26, -91.85) mm, rotated rx -152.51 ry -6.42 rz -112.51 deg; joints [14.574, -21.76, 71.222, 215.929, 101.714, 37.562, 26.033]
  MoveL 2567 to (-44.66, 46.35, -91.8) mm, rotated rx -152.51 ry -6.42 rz -112.51 deg; joints [14.587, -21.758, 71.208, 215.936, 101.709, 37.547, 26.033]
  MoveL 2568 to (-45.11, 46.46, -91.76) mm, rotated rx -152.51 ry -6.42 rz -112.51 deg; joints [14.6, -21.758, 71.194, 215.943, 101.702, 37.531, 26.033]
  MoveL 2569 to (-45.59, 46.59, -91.74) mm, rotated rx -152.51 ry -6.42 rz -112.51 deg; joints [14.615, -21.76, 71.18, 215.951, 101.696, 37.515, 26.033]
  MoveL 2570 to (-46.08, 46.73, -91.73) mm, rotated rx -152.51 ry -6.42 rz -112.51 deg; joints [14.629, -21.762, 71.167, 215.958, 101.689, 37.498, 26.033]
  MoveL 2571 to (-46.56, 46.86, -91.71) mm, rotated rx -152.51 ry -6.42 rz -112.51 deg; joints [14.643, -21.764, 71.154, 215.966, 101.682, 37.481, 26.033]
  MoveL 2572 to (-47.02, 46.97, -91.68) mm, rotated rx -152.51 ry -6.42 rz -112.51 deg; joints [14.657, -21.764, 71.14, 215.973, 101.676, 37.465, 26.033]
  MoveL 2573 to (-47.45, 47.05, -91.62) mm, rotated rx -152.51 ry -6.42 rz -112.51 deg; joints [14.67, -21.762, 71.126, 215.98, 101.671, 37.451, 26.033]
  MoveL 2574 to (-47.9, 47.14, -91.57) mm, rotated rx -152.51 ry -6.42 rz -112.51 deg; joints [14.683, -21.761, 71.111, 215.987, 101.665, 37.436, 26.033]
  MoveL 2575 to (-49.29, 47.48, -91.48) mm, rotated rx -152.51 ry -6.42 rz -112.51 deg; joints [14.725, -21.763, 71.071, 216.009, 101.647, 37.388, 26.033]
  MoveL 2576 to (-50.39, 47.9, -91.61) mm, rotated rx -152.51 ry -6.42 rz -112.51 deg; joints [14.756, -21.779, 71.051, 216.025, 101.629, 37.349, 26.033]
  MoveL 2577 to (-51.19, 48.4, -91.95) mm, rotated rx -152.51 ry -6.42 rz -112.51 deg; joints [14.777, -21.81, 71.05, 216.034, 101.612, 37.32, 26.033]
  MoveL 2578 to (-51.48, 48.68, -92.2) mm, rotated rx -152.51 ry -6.42 rz -112.51 deg; joints [14.783, -21.83, 71.058, 216.037, 101.604, 37.308, 26.033]
  MoveL 2579 to (-51.7, 48.98, -92.5) mm, rotated rx -152.51 ry -6.42 rz -112.51 deg; joints [14.787, -21.854, 71.07, 216.038, 101.597, 37.299, 26.033]
  MoveL 2580 to (-51.9, 49.63, -93.25) mm, rotated rx -152.51 ry -6.42 rz -112.51 deg; joints [14.787, -21.912, 71.11, 216.036, 101.582, 37.288, 26.033]
  MoveL 2581 to (-51.81, 50.37, -94.22) mm, rotated rx -152.51 ry -6.42 rz -112.51 deg; joints [14.776, -21.985, 71.17, 216.027, 101.567, 37.287, 26.033]
  MoveL 2582 to (-50.72, 52.06, -96.79) mm, rotated rx -152.51 ry -6.42 rz -112.51 deg; joints [14.724, -22.171, 71.35, 215.992, 101.542, 37.311, 26.033]
  MoveL 2583 to (-48.89, 53.52, -99.4) mm, rotated rx -152.51 ry -6.42 rz -112.51 deg; joints [14.649, -22.357, 71.554, 215.946, 101.528, 37.362, 26.033]
  MoveL 2584 to (-47.86, 53.96, -100.42) mm, rotated rx -152.51 ry -6.42 rz -112.51 deg; joints [14.611, -22.428, 71.645, 215.924, 101.53, 37.395, 26.033]
  MoveL 2585 to (-46.75, 54.2, -101.26) mm, rotated rx -152.51 ry -6.42 rz -112.51 deg; joints [14.572, -22.484, 71.728, 215.902, 101.537, 37.432, 26.033]
  MoveL 2586 to (-45.56, 54.25, -101.92) mm, rotated rx -152.51 ry -6.42 rz -112.51 deg; joints [14.533, -22.526, 71.804, 215.88, 101.549, 37.474, 26.033]
  MoveL 2587 to (-44.3, 54.11, -102.38) mm, rotated rx -152.51 ry -6.42 rz -112.51 deg; joints [14.493, -22.553, 71.873, 215.859, 101.568, 37.52, 26.033]
  MoveL 2588 to (-42.96, 53.77, -102.66) mm, rotated rx -152.51 ry -6.42 rz -112.51 deg; joints [14.452, -22.566, 71.935, 215.839, 101.592, 37.571, 26.033]
  MoveL 2589 to (-41.55, 53.23, -102.76) mm, rotated rx -152.51 ry -6.42 rz -112.51 deg; joints [14.411, -22.565, 71.989, 215.819, 101.621, 37.627, 26.033]
  MoveL 2590 to (-38.65, 51.97, -102.76) mm, rotated rx -152.51 ry -6.42 rz -112.51 deg; joints [14.329, -22.547, 72.089, 215.779, 101.686, 37.741, 26.033]
  MoveL 2591 to (-38.13, 51.75, -102.77) mm, rotated rx -152.51 ry -6.42 rz -112.51 deg; joints [14.314, -22.545, 72.108, 215.772, 101.697, 37.762, 26.033]
  MoveL 2592 to (-37.56, 51.53, -102.81) mm, rotated rx -152.51 ry -6.42 rz -112.51 deg; joints [14.297, -22.544, 72.13, 215.764, 101.709, 37.785, 26.033]
  MoveL 2593 to (-36.84, 51.28, -102.9) mm, rotated rx -152.51 ry -6.42 rz -112.51 deg; joints [14.276, -22.546, 72.16, 215.754, 101.724, 37.813, 26.033]
  MoveL 2594 to (-36.26, 51.06, -102.94) mm, rotated rx -152.51 ry -6.42 rz -112.51 deg; joints [14.259, -22.545, 72.182, 215.746, 101.737, 37.835, 26.033]
  MoveL 2595 to (-35.76, 50.85, -102.96) mm, rotated rx -152.51 ry -6.42 rz -112.51 deg; joints [14.245, -22.543, 72.201, 215.739, 101.747, 37.855, 26.033]
  MoveL 2596 to (-35.29, 50.65, -102.96) mm, rotated rx -152.51 ry -6.42 rz -112.51 deg; joints [14.232, -22.541, 72.217, 215.732, 101.758, 37.874, 26.033]
  MoveL 2597 to (-34.87, 50.48, -102.98) mm, rotated rx -152.51 ry -6.42 rz -112.51 deg; joints [14.219, -22.539, 72.232, 215.726, 101.767, 37.89, 26.033]
  MoveL 2598 to (-32.98, 49.67, -102.99) mm, rotated rx -152.51 ry -6.42 rz -112.51 deg; joints [14.165, -22.527, 72.297, 215.7, 101.808, 37.965, 26.033]
  MoveL 2599 to (-32.5, 49.48, -103.02) mm, rotated rx -152.51 ry -6.42 rz -112.51 deg; joints [14.151, -22.527, 72.315, 215.694, 101.818, 37.983, 26.033]
  MoveL 2600 to (-32.05, 49.33, -103.08) mm, rotated rx -152.51 ry -6.42 rz -112.51 deg; joints [14.138, -22.528, 72.333, 215.687, 101.827, 38.001, 26.033]
  MoveL 2601 to (-31.61, 49.2, -103.15) mm, rotated rx -152.51 ry -6.42 rz -112.51 deg; joints [14.125, -22.53, 72.352, 215.68, 101.836, 38.017, 26.033]
  MoveL 2602 to (-31.14, 49.08, -103.21) mm, rotated rx -152.51 ry -6.42 rz -112.51 deg; joints [14.111, -22.531, 72.369, 215.673, 101.843, 38.034, 26.033]
  MoveL 2603 to (-30.6, 48.96, -103.24) mm, rotated rx -152.51 ry -6.42 rz -112.51 deg; joints [14.095, -22.53, 72.383, 215.664, 101.849, 38.052, 26.033]
  MoveL 2604 to (-29.93, 48.91, -103.25) mm, rotated rx -152.51 ry -6.42 rz -112.51 deg; joints [14.074, -22.526, 72.39, 215.652, 101.85, 38.07, 26.033]
  MoveL 2605 to (-29.16, 48.92, -103.25) mm, rotated rx -152.51 ry -6.42 rz -112.51 deg; joints [14.049, -22.521, 72.392, 215.637, 101.847, 38.087, 26.033]
  MoveL 2606 to (-30.88, 49.82, -104.8) mm, rotated rx -152.51 ry -6.42 rz -112.51 deg; joints [14.093, -22.65, 72.498, 215.663, 101.845, 38.05, 26.033]
  MoveL 2607 to (-28.56, 50.27, -104.94) mm, rotated rx -152.51 ry -6.42 rz -112.51 deg; joints [14.016, -22.643, 72.49, 215.612, 101.816, 38.091, 26.033]
  MoveL 2608 to (-26.36, 50.69, -105.05) mm, rotated rx -152.51 ry -6.42 rz -112.51 deg; joints [13.944, -22.634, 72.481, 215.565, 101.788, 38.129, 26.033]
  MoveL 2609 to (-24.24, 51.1, -105.21) mm, rotated rx -152.51 ry -6.42 rz -112.51 deg; joints [13.874, -22.631, 72.477, 215.519, 101.762, 38.166, 26.033]
  MoveL 2610 to (-22.15, 51.51, -105.32) mm, rotated rx -152.51 ry -6.42 rz -112.51 deg; joints [13.806, -22.623, 72.468, 215.474, 101.735, 38.203, 26.033]
  MoveL 2611 to (-20.05, 51.91, -105.42) mm, rotated rx -152.51 ry -6.42 rz -112.51 deg; joints [13.737, -22.615, 72.459, 215.429, 101.708, 38.239, 26.033]
  MoveL 2612 to (-17.95, 52.32, -105.64) mm, rotated rx -152.51 ry -6.42 rz -112.51 deg; joints [13.667, -22.616, 72.461, 215.383, 101.683, 38.277, 26.033]
  MoveL 2613 to (-15.86, 52.73, -105.87) mm, rotated rx -152.51 ry -6.42 rz -112.51 deg; joints [13.598, -22.616, 72.464, 215.338, 101.659, 38.315, 26.033]
  MoveL 2614 to (-13.76, 53.12, -105.98) mm, rotated rx -152.51 ry -6.42 rz -112.51 deg; joints [13.529, -22.608, 72.455, 215.293, 101.633, 38.352, 26.033]
  MoveL 2615 to (-11.66, 53.5, -105.98) mm, rotated rx -152.51 ry -6.42 rz -112.51 deg; joints [13.46, -22.592, 72.434, 215.247, 101.603, 38.386, 26.033]
